LIN {X 0,Y 418.019,Z 608.172,A -85,B 0,C 180,E1 -10181.64,E2 -10181.64} C_VEL
LIN {X 0,Y 418.454,Z 601.286,A -85,B 0,C 180,E1 -10183.199,E2 -10183.199} C_VEL
LIN {X 0,Y 419.357,Z 591.379,A -85,B 0,C 180,E1 -10185.056,E2 -10185.056} C_VEL
LIN {X 0,Y 420.272,Z 581.997,A -85,B 0,C 180,E1 -10186.516,E2 -10186.516} C_VEL
LIN {X 0,Y 421.372,Z 571.359,A -85,B 0,C 180,E1 -10187.916,E2 -10187.916} C_VEL
LIN {X 0,Y 422.401,Z 559.979,A -85,B 0,C 180,E1 -10189.184,E2 -10189.184} C_VEL
LIN {X 0,Y 423.71,Z 546.942,A -85,B 0,C 180,E1 -10190.385,E2 -10190.385} C_VEL
LIN {X 0,Y 424.81,Z 534.302,A -85,B 0,C 180,E1 -10191.344,E2 -10191.344} C_VEL
LIN {X 0,Y 425.878,Z 520.707,A -85,B 0,C 180,E1 -10192.178,E2 -10192.178} C_VEL
LIN {X 0,Y 426.789,Z 506.169,A -85,B 0,C 180,E1 -10192.872,E2 -10192.872} C_VEL
LIN {X 0,Y 427.616,Z 490.972,A -85,B 0,C 180,E1 -10193.392,E2 -10193.392} C_VEL
LIN {X 0,Y 428.088,Z 474.732,A -85,B 0,C 180,E1 -10193.749,E2 -10193.749} C_VEL
LIN {X 0,Y 430.248,Z 350.197,A -85,B 0,C 180,E1 -10195.915,E2 -10195.915} C_VEL
LIN {X 0,Y 424.062,Z 318.078,A -85,B 0,C 180,E1 -10196.936,E2 -10196.936} C_VEL
LIN {X 0,Y 424.465,Z 312.588,A -85,B 0,C 180,E1 -10197.843,E2 -10197.843} C_VEL
LIN {X 0,Y 422.332,Z 302.144,A -85,B 0,C 180,E1 -10199.785,E2 -10199.785} C_VEL
LIN {X 0,Y 418.237,Z 286.016,A -85,B 0,C 180,E1 -10202.984,E2 -10202.984} C_VEL
LIN {X 0,Y 418.242,Z 286.015,A -85,B 0,C 180,E1 -10206.236,E2 -10206.236} C_VEL
LIN {X 0,Y 418.199,Z 286.022,A -85,B 0,C 180,E1 -10209.687,E2 -10209.687} C_VEL
LIN {X 0,Y 418.208,Z 286.015,A -85,B 0,C 180,E1 -10212.317,E2 -10212.317} C_VEL
LIN {X 0,Y 418.235,Z 286.012,A -85,B 0,C 180,E1 -10215.107,E2 -10215.107} C_VEL
LIN {X 0,Y 418.22,Z 286.015,A -85,B 0,C 180,E1 -10217.763,E2 -10217.763} C_VEL
LIN {X 0,Y 418.233,Z 286.01,A -85,B 0,C 180,E1 -10221.555,E2 -10221.555} C_VEL
LIN {X 0,Y 418.248,Z 286.005,A -85,B 0,C 180,E1 -10225.157,E2 -10225.157} C_VEL
LIN {X 0,Y 418.242,Z 286.009,A -85,B 0,C 180,E1 -10227.47,E2 -10227.47} C_VEL
LIN {X 0,Y 418.26,Z 286.007,A -85,B 0,C 180,E1 -10230.896,E2 -10230.896} C_VEL
LIN {X 0,Y 418.215,Z 286.019,A -85,B 0,C 180,E1 -10234.091,E2 -10234.091} C_VEL
LIN {X 0,Y 418.225,Z 286.012,A -85,B 0,C 180,E1 -10237.262,E2 -10237.262} C_VEL
LIN {X 0,Y 418.28,Z 286.004,A -85,B 0,C 180,E1 -10240.363,E2 -10240.363} C_VEL
LIN {X 0,Y 418.312,Z 286.006,A -85,B 0,C 180,E1 -10243.403,E2 -10243.403} C_VEL
LIN {X 0,Y 418.342,Z 285.979,A -85,B 0,C 180,E1 -10246.999,E2 -10246.999} C_VEL
LIN {X 0,Y 418.313,Z 285.998,A -85,B 0,C 180,E1 -10250.327,E2 -10250.327} C_VEL
LIN {X 0,Y 418.435,Z 285.988,A -85,B 0,C 180,E1 -10253.247,E2 -10253.247} C_VEL
LIN {X 0,Y 418.302,Z 285.996,A -85,B 0,C 180,E1 -10255.18,E2 -10255.18} C_VEL
LIN {X 0,Y 418.521,Z 285.966,A -85,B 0,C 180,E1 -10258.074,E2 -10258.074} C_VEL
LIN {X 0,Y 418.397,Z 285.989,A -85,B 0,C 180,E1 -10260.961,E2 -10260.961} C_VEL
LIN {X 0,Y 418.469,Z 285.98,A -85,B 0,C 180,E1 -10262.886,E2 -10262.886} C_VEL
LIN {X 0,Y 418.403,Z 285.965,A -85,B 0,C 180,E1 -10266.751,E2 -10266.751} C_VEL
LIN {X 0,Y 418.315,Z 286.001,A -85,B 0,C 180,E1 -10269.67,E2 -10269.67} C_VEL
LIN {X 0,Y 418.337,Z 285.999,A -85,B 0,C 180,E1 -10272.998,E2 -10272.998} C_VEL
LIN {X 0,Y 418.295,Z 285.982,A -85,B 0,C 180,E1 -10276.73,E2 -10276.73} C_VEL
LIN {X 0,Y 418.259,Z 286.005,A -85,B 0,C 180,E1 -10279.788,E2 -10279.788} C_VEL
LIN {X 0,Y 418.216,Z 286.013,A -85,B 0,C 180,E1 -10282.735,E2 -10282.735} C_VEL
LIN {X 0,Y 418.205,Z 285.997,A -85,B 0,C 180,E1 -10285.906,E2 -10285.906} C_VEL
LIN {X 0,Y 418.244,Z 286,A -85,B 0,C 180,E1 -10289.161,E2 -10289.161} C_VEL
LIN {X 0,Y 418.229,Z 286.011,A -85,B 0,C 180,E1 -10292.527,E2 -10292.527} C_VEL
LIN {X 0,Y 418.236,Z 286.006,A -85,B 0,C 180,E1 -10294.84,E2 -10294.84} C_VEL
LIN {X 0,Y 418.223,Z 286.002,A -85,B 0,C 180,E1 -10298.442,E2 -10298.442} C_VEL
LIN {X 0,Y 418.208,Z 286.013,A -85,B 0,C 180,E1 -10302.234,E2 -10302.234} C_VEL
LIN {X 0,Y 418.219,Z 286.001,A -85,B 0,C 180,E1 -10305.107,E2 -10305.107} C_VEL
LIN {X 0,Y 418.218,Z 286.012,A -85,B 0,C 180,E1 -10307.765,E2 -10307.765} C_VEL
LIN {X 0,Y 418.229,Z 286.015,A -85,B 0,C 180,E1 -10310.62,E2 -10310.62} C_VEL
LIN {X 0,Y 418.226,Z 286.004,A -85,B 0,C 180,E1 -10313.975,E2 -10313.975} C_VEL
LIN {X 0,Y 418.24,Z 286.012,A -85,B 0,C 180,E1 -10317.155,E2 -10317.155} C_VEL
LIN {X 0,Y 418.251,Z 286.006,A -85,B 0,C 180,E1 -10320.895,E2 -10320.895} C_VEL
LIN {X 0,Y 418.25,Z 286.006,A -85,B 0,C 180,E1 -10324.095,E2 -10324.095} C_VEL
LIN {X 0,Y 418.214,Z 286.016,A -85,B 0,C 180,E1 -10327.263,E2 -10327.263} C_VEL
LIN {X 0,Y 418.265,Z 286.004,A -85,B 0,C 180,E1 -10330.363,E2 -10330.363} C_VEL
LIN {X 0,Y 418.299,Z 285.999,A -85,B 0,C 180,E1 -10333.404,E2 -10333.404} C_VEL
LIN {X 0,Y 418.338,Z 285.999,A -85,B 0,C 180,E1 -10336.993,E2 -10336.993} C_VEL
LIN {X 0,Y 418.342,Z 285.997,A -85,B 0,C 180,E1 -10340.328,E2 -10340.328} C_VEL
LIN {X 0,Y 418.471,Z 285.983,A -85,B 0,C 180,E1 -10343.248,E2 -10343.248} C_VEL
LIN {X 0,Y 418.319,Z 286.004,A -85,B 0,C 180,E1 -10345.181,E2 -10345.181} C_VEL
LIN {X 0,Y 418.524,Z 285.974,A -85,B 0,C 180,E1 -10348.075,E2 -10348.075} C_VEL
LIN {X 0,Y 418.534,Z 285.982,A -85,B 0,C 180,E1 -10350.601,E2 -10350.601} C_VEL
LIN {X 0,Y 420.885,Z 296.753,A -85,B 0,C 180,E1 -10352.944,E2 -10352.944} C_VEL
LIN {X 0,Y 428.881,Z 316.026,A -85,B 0,C 180,E1 -10353.834,E2 -10353.834} C_VEL
LIN {X 0,Y 430.579,Z 324.35,A -85,B 0,C 180,E1 -10354.097,E2 -10354.097} C_VEL
LIN {X 0,Y 430.008,Z 354.65,A -85,B 0,C 180,E1 -10354.626,E2 -10354.626} C_VEL
LIN {X 0,Y 429.344,Z 360.497,A -85,B 0,C 180,E1 -10354.695,E2 -10354.695} C_VEL
LIN {X 0,Y 423.7,Z 379.54,A -85,B 0,C 180,E1 -10354.705,E2 -10354.705} C_VEL
LIN {X 0,Y 422.973,Z 385.393,A -85,B 0,C 180,E1 -10354.77,E2 -10354.77} C_VEL
LIN {X 0,Y 421.513,Z 462.7,A -85,B 0,C 180,E1 -10356.161,E2 -10356.161} C_VEL
LIN {X 0,Y 420.889,Z 477.855,A -85,B 0,C 180,E1 -10356.622,E2 -10356.622} C_VEL
LIN {X 0,Y 420.031,Z 492.733,A -85,B 0,C 180,E1 -10357.269,E2 -10357.269} C_VEL
LIN {X 0,Y 419.023,Z 507.308,A -85,B 0,C 180,E1 -10358.113,E2 -10358.113} C_VEL
LIN {X 0,Y 417.877,Z 520.501,A -85,B 0,C 180,E1 -10359.071,E2 -10359.071} C_VEL
LIN {X 0,Y 416.658,Z 533.182,A -85,B 0,C 180,E1 -10360.201,E2 -10360.201} C_VEL
LIN {X 0,Y 415.406,Z 545.864,A -85,B 0,C 180,E1 -10361.573,E2 -10361.573} C_VEL
LIN {X 0,Y 414.269,Z 556.742,A -85,B 0,C 180,E1 -10362.989,E2 -10362.989} C_VEL
LIN {X 0,Y 413.218,Z 566.322,A -85,B 0,C 180,E1 -10364.468,E2 -10364.468} C_VEL
LIN {X 0,Y 412.281,Z 575.139,A -85,B 0,C 180,E1 -10366.081,E2 -10366.081} C_VEL
LIN {X 0,Y 411.458,Z 583.427,A -85,B 0,C 180,E1 -10367.905,E2 -10367.905} C_VEL
LIN {X 0,Y 410.868,Z 590.526,A -85,B 0,C 180,E1 -10369.823,E2 -10369.823} C_VEL
LIN {X 0,Y 410.453,Z 595.842,A -85,B 0,C 180,E1 -10371.6,E2 -10371.6} C_VEL
LIN {X 0,Y 410.153,Z 600.738,A -85,B 0,C 180,E1 -10373.744,E2 -10373.744} C_VEL
LIN {X 0,Y 409.89,Z 603.462,A -85,B 0,C 180,E1 -10375.381,E2 -10375.381} C_VEL
LIN {X 0,Y 409.738,Z 605.849,A -85,B 0,C 180,E1 -10377.587,E2 -10377.587} C_VEL
LIN {X 0,Y 409.691,Z 606.635,A -85,B 0,C 180,E1 -10378.975,E2 -10378.975} C_VEL
LIN {X 0,Y 409.739,Z 606.704,A -85,B 0,C 180,E1 -10380.968,E2 -10380.968} C_VEL
LIN {X 0,Y 409.784,Z 605.724,A -85,B 0,C 180,E1 -10382.825,E2 -10382.825} C_VEL
LIN {X 0,Y 409.892,Z 603.843,A -85,B 0,C 180,E1 -10384.617,E2 -10384.617} C_VEL
LIN {X 0,Y 410.153,Z 601.026,A -85,B 0,C 180,E1 -10386.36,E2 -10386.36} C_VEL
LIN {X 0,Y 410.415,Z 597.353,A -85,B 0,C 180,E1 -10388.057,E2 -10388.057} C_VEL
LIN {X 0,Y 410.855,Z 591.79,A -85,B 0,C 180,E1 -10390.053,E2 -10390.053} C_VEL
LIN {X 0,Y 411.509,Z 584.791,A -85,B 0,C 180,E1 -10392.028,E2 -10392.028} C_VEL
LIN {X 0,Y 412.221,Z 577.732,A -85,B 0,C 180,E1 -10393.667,E2 -10393.667} C_VEL
LIN {X 0,Y 413.095,Z 569.526,A -85,B 0,C 180,E1 -10395.257,E2 -10395.257} C_VEL
LIN {X 0,Y 414.171,Z 559.721,A -85,B 0,C 180,E1 -10396.856,E2 -10396.856} C_VEL
LIN {X 0,Y 415.357,Z 549.189,A -85,B 0,C 180,E1 -10398.296,E2 -10398.296} C_VEL
LIN {X 0,Y 416.685,Z 536.811,A -85,B 0,C 180,E1 -10399.709,E2 -10399.709} C_VEL
LIN {X 0,Y 417.964,Z 524.647,A -85,B 0,C 180,E1 -10400.856,E2 -10400.856} C_VEL
LIN {X 0,Y 419.116,Z 511.674,A -85,B 0,C 180,E1 -10401.868,E2 -10401.868} C_VEL
LIN {X 0,Y 420.267,Z 497.228,A -85,B 0,C 180,E1 -10402.766,E2 -10402.766} C_VEL
LIN {X 0,Y 421.236,Z 482.096,A -85,B 0,C 180,E1 -10403.483,E2 -10403.483} C_VEL
LIN {X 0,Y 421.955,Z 466.599,A -85,B 0,C 180,E1 -10404.006,E2 -10404.006} C_VEL
LIN {X 0,Y 422.457,Z 446.837,A -85,B 0,C 180,E1 -10404.418,E2 -10404.418} C_VEL
LIN {X 0,Y 424.854,Z 325.118,A -85,B 0,C 180,E1 -10406.598,E2 -10406.598} C_VEL
LIN {X 0,Y 423.221,Z 318.56,A -85,B 0,C 180,E1 -10406.844,E2 -10406.844} C_VEL
LIN {X 0,Y 415.127,Z 300.427,A -85,B 0,C 180,E1 -10407.818,E2 -10407.818} C_VEL
LIN {X 0,Y 413.924,Z 297.657,A -85,B 0,C 180,E1 -10408.001,E2 -10408.001} C_VEL
LIN {X 0,Y 411.237,Z 286.889,A -85,B 0,C 180,E1 -10410.516,E2 -10410.516} C_VEL
LIN {X 0,Y 411.222,Z 286.886,A -85,B 0,C 180,E1 -10413.62,E2 -10413.62} C_VEL
LIN {X 0,Y 411.188,Z 286.896,A -85,B 0,C 180,E1 -10416.854,E2 -10416.854} C_VEL
LIN {X 0,Y 411.2,Z 286.89,A -85,B 0,C 180,E1 -10420.052,E2 -10420.052} C_VEL
LIN {X 0,Y 411.249,Z 286.886,A -85,B 0,C 180,E1 -10423.133,E2 -10423.133} C_VEL
LIN {X 0,Y 411.291,Z 286.879,A -85,B 0,C 180,E1 -10426.898,E2 -10426.898} C_VEL
LIN {X 0,Y 411.279,Z 286.878,A -85,B 0,C 180,E1 -10430.163,E2 -10430.163} C_VEL
LIN {X 0,Y 411.445,Z 286.859,A -85,B 0,C 180,E1 -10433.135,E2 -10433.135} C_VEL
LIN {X 0,Y 411.295,Z 286.88,A -85,B 0,C 180,E1 -10435.101,E2 -10435.101} C_VEL
LIN {X 0,Y 411.5,Z 286.85,A -85,B 0,C 180,E1 -10438.044,E2 -10438.044} C_VEL
LIN {X 0,Y 411.629,Z 286.833,A -85,B 0,C 180,E1 -10440.002,E2 -10440.002} C_VEL
LIN {X 0,Y 411.442,Z 286.86,A -85,B 0,C 180,E1 -10442.939,E2 -10442.939} C_VEL
LIN {X 0,Y 411.423,Z 286.862,A -85,B 0,C 180,E1 -10446.869,E2 -10446.869} C_VEL
LIN {X 0,Y 411.28,Z 286.877,A -85,B 0,C 180,E1 -10449.84,E2 -10449.84} C_VEL
LIN {X 0,Y 411.297,Z 286.875,A -85,B 0,C 180,E1 -10453.105,E2 -10453.105} C_VEL
LIN {X 0,Y 411.249,Z 286.88,A -85,B 0,C 180,E1 -10456.89,E2 -10456.89} C_VEL
LIN {X 0,Y 411.223,Z 286.884,A -85,B 0,C 180,E1 -10459.988,E2 -10459.988} C_VEL
LIN {X 0,Y 411.179,Z 286.888,A -85,B 0,C 180,E1 -10463.15,E2 -10463.15} C_VEL
LIN {X 0,Y 411.167,Z 286.891,A -85,B 0,C 180,E1 -10466.387,E2 -10466.387} C_VEL
LIN {X 0,Y 411.19,Z 286.886,A -85,B 0,C 180,E1 -10469.715,E2 -10469.715} C_VEL
LIN {X 0,Y 411.199,Z 286.886,A -85,B 0,C 180,E1 -10473.158,E2 -10473.158} C_VEL
LIN {X 0,Y 411.183,Z 286.888,A -85,B 0,C 180,E1 -10476.553,E2 -10476.553} C_VEL
LIN {X 0,Y 411.163,Z 286.89,A -85,B 0,C 180,E1 -10479.721,E2 -10479.721} C_VEL
LIN {X 0,Y 411.158,Z 286.892,A -85,B 0,C 180,E1 -10483.137,E2 -10483.137} C_VEL
LIN {X 0,Y 411.16,Z 286.894,A -85,B 0,C 180,E1 -10485.883,E2 -10485.883} C_VEL
LIN {X 0,Y 411.155,Z 286.894,A -85,B 0,C 180,E1 -10489.494,E2 -10489.494} C_VEL
LIN {X 0,Y 411.179,Z 286.892,A -85,B 0,C 180,E1 -10492.026,E2 -10492.026} C_VEL
LIN {X 0,Y 411.202,Z 286.885,A -85,B 0,C 180,E1 -10495.667,E2 -10495.667} C_VEL
LIN {X 0,Y 411.239,Z 286.989,A -85,B 0,C 180,E1 -10496.262,E2 -10496.262} C_VEL
LIN {X 0,Y 415.258,Z 302.312,A -85,B 0,C 180,E1 -10499.488,E2 -10499.488} C_VEL
LIN {X 0,Y 417.681,Z 313.276,A -85,B 0,C 180,E1 -10501.653,E2 -10501.653} C_VEL
LIN {X 0,Y 417.681,Z 317.189,A -85,B 0,C 180,E1 -10502.344,E2 -10502.344} C_VEL
LIN {X 0,Y 422.839,Z 342.545,A -85,B 0,C 180,E1 -10503.237,E2 -10503.237} C_VEL
LIN {X 0,Y 424.557,Z 352.473,A -85,B 0,C 180,E1 -10503.551,E2 -10503.551} C_VEL
LIN {X 0,Y 421.834,Z 483.858,A -85,B 0,C 180,E1 -10505.91,E2 -10505.91} C_VEL
LIN {X 0,Y 421.04,Z 499.798,A -85,B 0,C 180,E1 -10506.385,E2 -10506.385} C_VEL
LIN {X 0,Y 420.117,Z 514.266,A -85,B 0,C 180,E1 -10507.007,E2 -10507.007} C_VEL
LIN {X 0,Y 418.915,Z 528.72,A -85,B 0,C 180,E1 -10507.824,E2 -10507.824} C_VEL
LIN {X 0,Y 417.691,Z 542.21,A -85,B 0,C 180,E1 -10508.793,E2 -10508.793} C_VEL
LIN {X 0,Y 416.259,Z 555.968,A -85,B 0,C 180,E1 -10510.008,E2 -10510.008} C_VEL
LIN {X 0,Y 415.097,Z 567.363,A -85,B 0,C 180,E1 -10511.236,E2 -10511.236} C_VEL
LIN {X 0,Y 413.886,Z 578.907,A -85,B 0,C 180,E1 -10512.714,E2 -10512.714} C_VEL
LIN {X 0,Y 412.782,Z 588.63,A -85,B 0,C 180,E1 -10514.193,E2 -10514.193} C_VEL
LIN {X 0,Y 411.805,Z 598.188,A -85,B 0,C 180,E1 -10515.926,E2 -10515.926} C_VEL
LIN {X 0,Y 411.112,Z 606.159,A -85,B 0,C 180,E1 -10517.662,E2 -10517.662} C_VEL
LIN {X 0,Y 410.504,Z 613.606,A -85,B 0,C 180,E1 -10519.645,E2 -10519.645} C_VEL
LIN {X 0,Y 410.2,Z 619.523,A -85,B 0,C 180,E1 -10521.627,E2 -10521.627} C_VEL
LIN {X 0,Y 410.012,Z 623.044,A -85,B 0,C 180,E1 -10523.109,E2 -10523.109} C_VEL
LIN {X 0,Y 409.927,Z 626.598,A -85,B 0,C 180,E1 -10525.083,E2 -10525.083} C_VEL
LIN {X 0,Y 409.906,Z 628.934,A -85,B 0,C 180,E1 -10527.052,E2 -10527.052} C_VEL
LIN {X 0,Y 409.935,Z 630.103,A -85,B 0,C 180,E1 -10529.018,E2 -10529.018} C_VEL
LIN {X 0,Y 409.935,Z 630.105,A -85,B 0,C 180,E1 -10530.983,E2 -10530.983} C_VEL
LIN {X 0,Y 409.907,Z 628.9,A -85,B 0,C 180,E1 -10532.949,E2 -10532.949} C_VEL
LIN {X 0,Y 409.935,Z 626.527,A -85,B 0,C 180,E1 -10534.918,E2 -10534.918} C_VEL
LIN {X 0,Y 410.051,Z 622.935,A -85,B 0,C 180,E1 -10536.891,E2 -10536.891} C_VEL
LIN {X 0,Y 410.241,Z 618.028,A -85,B 0,C 180,E1 -10538.87,E2 -10538.87} C_VEL
LIN {X 0,Y 410.674,Z 611.68,A -85,B 0,C 180,E1 -10540.851,E2 -10540.851} C_VEL
LIN {X 0,Y 411.254,Z 603.708,A -85,B 0,C 180,E1 -10542.836,E2 -10542.836} C_VEL
LIN {X 0,Y 412.049,Z 595.217,A -85,B 0,C 180,E1 -10544.571,E2 -10544.571} C_VEL
LIN {X 0,Y 412.824,Z 586.588,A -85,B 0,C 180,E1 -10546.06,E2 -10546.06} C_VEL
LIN {X 0,Y 414.02,Z 576.388,A -85,B 0,C 180,E1 -10547.536,E2 -10547.536} C_VEL
LIN {X 0,Y 415.067,Z 565.321,A -85,B 0,C 180,E1 -10548.895,E2 -10548.895} C_VEL
LIN {X 0,Y 416.3,Z 553.387,A -85,B 0,C 180,E1 -10550.119,E2 -10550.119} C_VEL
LIN {X 0,Y 417.551,Z 540.482,A -85,B 0,C 180,E1 -10551.215,E2 -10551.215} C_VEL
LIN {X 0,Y 418.753,Z 526.377,A -85,B 0,C 180,E1 -10552.186,E2 -10552.186} C_VEL
LIN {X 0,Y 419.881,Z 511.447,A -85,B 0,C 180,E1 -10552.986,E2 -10552.986} C_VEL
LIN {X 0,Y 420.719,Z 496.663,A -85,B 0,C 180,E1 -10553.575,E2 -10553.575} C_VEL
LIN {X 0,Y 421.368,Z 481.331,A -85,B 0,C 180,E1 -10553.988,E2 -10553.988} C_VEL
LIN {X 0,Y 423.834,Z 353.002,A -85,B 0,C 180,E1 -10556.261,E2 -10556.261} C_VEL
LIN {X 0,Y 423.233,Z 348.315,A -85,B 0,C 180,E1 -10556.388,E2 -10556.388} C_VEL
LIN {X 0,Y 417.369,Z 317.942,A -85,B 0,C 180,E1 -10557.375,E2 -10557.375} C_VEL
LIN {X 0,Y 417.596,Z 313.587,A -85,B 0,C 180,E1 -10558.114,E2 -10558.114} C_VEL
LIN {X 0,Y 414.758,Z 300.84,A -85,B 0,C 180,E1 -10560.553,E2 -10560.553} C_VEL
LIN {X 0,Y 411.192,Z 286.894,A -85,B 0,C 180,E1 -10563.369,E2 -10563.369} C_VEL
LIN {X 0,Y 411.188,Z 286.896,A -85,B 0,C 180,E1 -10566.742,E2 -10566.742} C_VEL
LIN {X 0,Y 411.169,Z 286.897,A -85,B 0,C 180,E1 -10569.719,E2 -10569.719} C_VEL
LIN {X 0,Y 411.162,Z 286.889,A -85,B 0,C 180,E1 -10573.134,E2 -10573.134} C_VEL
LIN {X 0,Y 411.164,Z 286.893,A -85,B 0,C 180,E1 -10575.881,E2 -10575.881} C_VEL
LIN {X 0,Y 411.148,Z 286.898,A -85,B 0,C 180,E1 -10578.773,E2 -10578.773} C_VEL
LIN {X 0,Y 411.18,Z 286.894,A -85,B 0,C 180,E1 -10582.024,E2 -10582.024} C_VEL
LIN {X 0,Y 411.2,Z 286.883,A -85,B 0,C 180,E1 -10585.123,E2 -10585.123} C_VEL
LIN {X 0,Y 411.163,Z 286.897,A -85,B 0,C 180,E1 -10588.001,E2 -10588.001} C_VEL
LIN {X 0,Y 411.174,Z 286.892,A -85,B 0,C 180,E1 -10591.405,E2 -10591.405} C_VEL
LIN {X 0,Y 411.186,Z 286.891,A -85,B 0,C 180,E1 -10594.94,E2 -10594.94} C_VEL
LIN {X 0,Y 411.2,Z 286.895,A -85,B 0,C 180,E1 -10597.912,E2 -10597.912} C_VEL
LIN {X 0,Y 411.214,Z 286.884,A -85,B 0,C 180,E1 -10601.05,E2 -10601.05} C_VEL
LIN {X 0,Y 411.247,Z 286.88,A -85,B 0,C 180,E1 -10604.13,E2 -10604.13} C_VEL
LIN {X 0,Y 411.297,Z 286.855,A -85,B 0,C 180,E1 -10607.164,E2 -10607.164} C_VEL
LIN {X 0,Y 411.268,Z 286.877,A -85,B 0,C 180,E1 -10610.159,E2 -10610.159} C_VEL
LIN {X 0,Y 411.384,Z 286.865,A -85,B 0,C 180,E1 -10613.13,E2 -10613.13} C_VEL
LIN {X 0,Y 411.274,Z 286.872,A -85,B 0,C 180,E1 -10615.097,E2 -10615.097} C_VEL
LIN {X 0,Y 411.49,Z 286.84,A -85,B 0,C 180,E1 -10618.041,E2 -10618.041} C_VEL
LIN {X 0,Y 411.497,Z 286.85,A -85,B 0,C 180,E1 -10621.956,E2 -10621.956} C_VEL
LIN {X 0,Y 411.348,Z 286.843,A -85,B 0,C 180,E1 -10626.445,E2 -10626.445} C_VEL
LIN {X 0,Y 411.276,Z 286.867,A -85,B 0,C 180,E1 -10628.845,E2 -10628.845} C_VEL
LIN {X 0,Y 411.271,Z 286.879,A -85,B 0,C 180,E1 -10631.831,E2 -10631.831} C_VEL
LIN {X 0,Y 411.237,Z 286.876,A -85,B 0,C 180,E1 -10634.852,E2 -10634.852} C_VEL
LIN {X 0,Y 411.23,Z 286.868,A -85,B 0,C 180,E1 -10637.914,E2 -10637.914} C_VEL
LIN {X 0,Y 411.185,Z 286.888,A -85,B 0,C 180,E1 -10641.033,E2 -10641.033} C_VEL
LIN {X 0,Y 411.178,Z 286.884,A -85,B 0,C 180,E1 -10644.216,E2 -10644.216} C_VEL
LIN {X 0,Y 411.133,Z 286.876,A -85,B 0,C 180,E1 -10647.484,E2 -10647.484} C_VEL
LIN {X 0,Y 411.183,Z 286.886,A -85,B 0,C 180,E1 -10649.712,E2 -10649.712} C_VEL
LIN {X 0,Y 411.191,Z 286.89,A -85,B 0,C 180,E1 -10653.155,E2 -10653.155} C_VEL
LIN {X 0,Y 411.177,Z 286.872,A -85,B 0,C 180,E1 -10656.551,E2 -10656.551} C_VEL
LIN {X 0,Y 411.155,Z 286.892,A -85,B 0,C 180,E1 -10659.719,E2 -10659.719} C_VEL
LIN {X 0,Y 411.149,Z 286.891,A -85,B 0,C 180,E1 -10663.134,E2 -10663.134} C_VEL
LIN {X 0,Y 411.15,Z 286.881,A -85,B 0,C 180,E1 -10665.88,E2 -10665.88} C_VEL
LIN {X 0,Y 411.144,Z 286.897,A -85,B 0,C 180,E1 -10668.771,E2 -10668.771} C_VEL
LIN {X 0,Y 411.175,Z 286.883,A -85,B 0,C 180,E1 -10672.025,E2 -10672.025} C_VEL
LIN {X 0,Y 411.188,Z 286.889,A -85,B 0,C 180,E1 -10675.665,E2 -10675.665} C_VEL
LIN {X 0,Y 411.172,Z 286.882,A -85,B 0,C 180,E1 -10679.151,E2 -10679.151} C_VEL
LIN {X 0,Y 411.249,Z 286.885,A -85,B 0,C 180,E1 -10682.698,E2 -10682.698} C_VEL
LIN {X 0,Y 411.194,Z 286.884,A -85,B 0,C 180,E1 -10685.783,E2 -10685.783} C_VEL
LIN {X 0,Y 411.179,Z 286.887,A -85,B 0,C 180,E1 -10688.965,E2 -10688.965} C_VEL
LIN {X 0,Y 411.234,Z 286.885,A -85,B 0,C 180,E1 -10692.084,E2 -10692.084} C_VEL
LIN {X 0,Y 411.244,Z 286.884,A -85,B 0,C 180,E1 -10695.147,E2 -10695.147} C_VEL
LIN {X 0,Y 411.283,Z 286.879,A -85,B 0,C 180,E1 -10698.167,E2 -10698.167} C_VEL
LIN {X 0,Y 411.422,Z 286.859,A -85,B 0,C 180,E1 -10702.188,E2 -10702.188} C_VEL
LIN {X 0,Y 411.452,Z 286.857,A -85,B 0,C 180,E1 -10704.117,E2 -10704.117} C_VEL
LIN {X 0,Y 411.493,Z 286.85,A -85,B 0,C 180,E1 -10708.042,E2 -10708.042} C_VEL
LIN {X 0,Y 411.583,Z 286.917,A -85,B 0,C 180,E1 -10710.275,E2 -10710.275} C_VEL
LIN {X 0,Y 413.798,Z 296.991,A -85,B 0,C 180,E1 -10712.464,E2 -10712.464} C_VEL
LIN {X 0,Y 422.753,Z 318.435,A -85,B 0,C 180,E1 -10713.484,E2 -10713.484} C_VEL
LIN {X 0,Y 424.172,Z 324.99,A -85,B 0,C 180,E1 -10713.701,E2 -10713.701} C_VEL
LIN {X 0,Y 422.973,Z 385.393,A -85,B 0,C 180,E1 -10714.77,E2 -10714.77} C_VEL
LIN {X 0,Y 422.255,Z 391.242,A -85,B 0,C 180,E1 -10714.835,E2 -10714.835} C_VEL
LIN {X 0,Y 416.637,Z 410.284,A -85,B 0,C 180,E1 -10714.849,E2 -10714.849} C_VEL
LIN {X 0,Y 415.934,Z 416.132,A -85,B 0,C 180,E1 -10714.917,E2 -10714.917} C_VEL
LIN {X 0,Y 415.006,Z 462.388,A -85,B 0,C 180,E1 -10715.77,E2 -10715.77} C_VEL
LIN {X 0,Y 414.361,Z 477.695,A -85,B 0,C 180,E1 -10716.237,E2 -10716.237} C_VEL
LIN {X 0,Y 413.461,Z 492.672,A -85,B 0,C 180,E1 -10716.894,E2 -10716.894} C_VEL
LIN {X 0,Y 412.448,Z 506.704,A -85,B 0,C 180,E1 -10717.711,E2 -10717.711} C_VEL
LIN {X 0,Y 411.177,Z 520.857,A -85,B 0,C 180,E1 -10718.749,E2 -10718.749} C_VEL
LIN {X 0,Y 409.817,Z 534.542,A -85,B 0,C 180,E1 -10719.999,E2 -10719.999} C_VEL
LIN {X 0,Y 408.552,Z 546.595,A -85,B 0,C 180,E1 -10721.34,E2 -10721.34} C_VEL
LIN {X 0,Y 407.239,Z 558.65,A -85,B 0,C 180,E1 -10722.964,E2 -10722.964} C_VEL
LIN {X 0,Y 406.076,Z 568.746,A -85,B 0,C 180,E1 -10724.598,E2 -10724.598} C_VEL
LIN {X 0,Y 405.06,Z 577.869,A -85,B 0,C 180,E1 -10726.376,E2 -10726.376} C_VEL
LIN {X 0,Y 404.281,Z 585.722,A -85,B 0,C 180,E1 -10728.234,E2 -10728.234} C_VEL
LIN {X 0,Y 403.752,Z 591.697,A -85,B 0,C 180,E1 -10729.963,E2 -10729.963} C_VEL
LIN {X 0,Y 403.315,Z 597.333,A -85,B 0,C 180,E1 -10731.988,E2 -10731.988} C_VEL
LIN {X 0,Y 403.095,Z 600.926,A -85,B 0,C 180,E1 -10733.64,E2 -10733.64} C_VEL
LIN {X 0,Y 402.742,Z 604.399,A -85,B 0,C 180,E1 -10735.864,E2 -10735.864} C_VEL
LIN {X 0,Y 402.697,Z 605.701,A -85,B 0,C 180,E1 -10737.124,E2 -10737.124} C_VEL
LIN {X 0,Y 402.584,Z 606.898,A -85,B 0,C 180,E1 -10739.261,E2 -10739.261} C_VEL
LIN {X 0,Y 402.632,Z 606.873,A -85,B 0,C 180,E1 -10741.212,E2 -10741.212} C_VEL
LIN {X 0,Y 402.7,Z 605.756,A -85,B 0,C 180,E1 -10743.106,E2 -10743.106} C_VEL
LIN {X 0,Y 402.867,Z 603.424,A -85,B 0,C 180,E1 -10745.146,E2 -10745.146} C_VEL
LIN {X 0,Y 403.136,Z 600.871,A -85,B 0,C 180,E1 -10746.689,E2 -10746.689} C_VEL
LIN {X 0,Y 403.505,Z 596.049,A -85,B 0,C 180,E1 -10748.829,E2 -10748.829} C_VEL
LIN {X 0,Y 403.968,Z 590.478,A -85,B 0,C 180,E1 -10750.721,E2 -10750.721} C_VEL
LIN {X 0,Y 404.711,Z 583.498,A -85,B 0,C 180,E1 -10752.628,E2 -10752.628} C_VEL
LIN {X 0,Y 405.604,Z 574.901,A -85,B 0,C 180,E1 -10754.544,E2 -10754.544} C_VEL
LIN {X 0,Y 406.742,Z 565.413,A -85,B 0,C 180,E1 -10756.282,E2 -10756.282} C_VEL
LIN {X 0,Y 407.897,Z 555.484,A -85,B 0,C 180,E1 -10757.805,E2 -10757.805} C_VEL
LIN {X 0,Y 409.259,Z 544.082,A -85,B 0,C 180,E1 -10759.269,E2 -10759.269} C_VEL
LIN {X 0,Y 410.653,Z 531.345,A -85,B 0,C 180,E1 -10760.627,E2 -10760.627} C_VEL
LIN {X 0,Y 412.046,Z 517.625,A -85,B 0,C 180,E1 -10761.82,E2 -10761.82} C_VEL
LIN {X 0,Y 413.242,Z 504.086,A -85,B 0,C 180,E1 -10762.768,E2 -10762.768} C_VEL
LIN {X 0,Y 414.345,Z 489.154,A -85,B 0,C 180,E1 -10763.586,E2 -10763.586} C_VEL
LIN {X 0,Y 415.232,Z 473.83,A -85,B 0,C 180,E1 -10764.203,E2 -10764.203} C_VEL
LIN {X 0,Y 415.815,Z 458.836,A -85,B 0,C 180,E1 -10764.61,E2 -10764.61} C_VEL
LIN {X 0,Y 418.589,Z 326.369,A -85,B 0,C 180,E1 -10767.031,E2 -10767.031} C_VEL
LIN {X 0,Y 417.293,Z 321.295,A -85,B 0,C 180,E1 -10767.23,E2 -10767.23} C_VEL
LIN {X 0,Y 409.485,Z 303.858,A -85,B 0,C 180,E1 -10768.195,E2 -10768.195} C_VEL
LIN {X 0,Y 406.781,Z 297.955,A -85,B 0,C 180,E1 -10768.566,E2 -10768.566} C_VEL
LIN {X 0,Y 404.175,Z 287.765,A -85,B 0,C 180,E1 -10771.009,E2 -10771.009} C_VEL
LIN {X 0,Y 404.168,Z 287.767,A -85,B 0,C 180,E1 -10774.235,E2 -10774.235} C_VEL
LIN {X 0,Y 404.155,Z 287.766,A -85,B 0,C 180,E1 -10777.51,E2 -10777.51} C_VEL
LIN {X 0,Y 404.151,Z 287.764,A -85,B 0,C 180,E1 -10780.709,E2 -10780.709} C_VEL
LIN {X 0,Y 404.207,Z 287.762,A -85,B 0,C 180,E1 -10783.85,E2 -10783.85} C_VEL
LIN {X 0,Y 404.269,Z 287.753,A -85,B 0,C 180,E1 -10786.94,E2 -10786.94} C_VEL
LIN {X 0,Y 404.244,Z 287.754,A -85,B 0,C 180,E1 -10789.99,E2 -10789.99} C_VEL
LIN {X 0,Y 404.392,Z 287.739,A -85,B 0,C 180,E1 -10793.014,E2 -10793.014} C_VEL
LIN {X 0,Y 404.268,Z 287.755,A -85,B 0,C 180,E1 -10795.015,E2 -10795.015} C_VEL
LIN {X 0,Y 404.468,Z 287.726,A -85,B 0,C 180,E1 -10798.01,E2 -10798.01} C_VEL
LIN {X 0,Y 404.599,Z 287.709,A -85,B 0,C 180,E1 -10800.002,E2 -10800.002} C_VEL
LIN {X 0,Y 404.4,Z 287.738,A -85,B 0,C 180,E1 -10802.99,E2 -10802.99} C_VEL
LIN {X 0,Y 404.373,Z 287.738,A -85,B 0,C 180,E1 -10806.989,E2 -10806.989} C_VEL
LIN {X 0,Y 404.241,Z 287.753,A -85,B 0,C 180,E1 -10811.027,E2 -10811.027} C_VEL
LIN {X 0,Y 404.201,Z 287.757,A -85,B 0,C 180,E1 -10814.09,E2 -10814.09} C_VEL
LIN {X 0,Y 404.195,Z 287.758,A -85,B 0,C 180,E1 -10817.194,E2 -10817.194} C_VEL
LIN {X 0,Y 404.156,Z 287.764,A -85,B 0,C 180,E1 -10820.353,E2 -10820.353} C_VEL
LIN {X 0,Y 404.141,Z 287.764,A -85,B 0,C 180,E1 -10823.578,E2 -10823.578} C_VEL
LIN {X 0,Y 404.113,Z 287.772,A -85,B 0,C 180,E1 -10826.884,E2 -10826.884} C_VEL
LIN {X 0,Y 404.137,Z 287.77,A -85,B 0,C 180,E1 -10830.287,E2 -10830.287} C_VEL
LIN {X 0,Y 404.132,Z 287.768,A -85,B 0,C 180,E1 -10833.815,E2 -10833.815} C_VEL
LIN {X 0,Y 404.125,Z 287.767,A -85,B 0,C 180,E1 -10836.875,E2 -10836.875} C_VEL
LIN {X 0,Y 404.113,Z 287.772,A -85,B 0,C 180,E1 -10840.076,E2 -10840.076} C_VEL
LIN {X 0,Y 404.137,Z 287.767,A -85,B 0,C 180,E1 -10843.083,E2 -10843.083} C_VEL
LIN {X 0,Y 404.117,Z 287.771,A -85,B 0,C 180,E1 -10845.923,E2 -10845.923} C_VEL
LIN {X 0,Y 404.099,Z 287.774,A -85,B 0,C 180,E1 -10848.634,E2 -10848.634} C_VEL
LIN {X 0,Y 404.135,Z 287.772,A -85,B 0,C 180,E1 -10851.497,E2 -10851.497} C_VEL
LIN {X 0,Y 404.18,Z 287.761,A -85,B 0,C 180,E1 -10854.985,E2 -10854.985} C_VEL
LIN {X 0,Y 404.182,Z 287.789,A -85,B 0,C 180,E1 -10855.742,E2 -10855.742} C_VEL
LIN {X 0,Y 408.316,Z 303.343,A -85,B 0,C 180,E1 -10859.113,E2 -10859.113} C_VEL
LIN {X 0,Y 410.827,Z 314.595,A -85,B 0,C 180,E1 -10861.381,E2 -10861.381} C_VEL
LIN {X 0,Y 411.081,Z 317.033,A -85,B 0,C 180,E1 -10861.841,E2 -10861.841} C_VEL
LIN {X 0,Y 416.364,Z 342.596,A -85,B 0,C 180,E1 -10862.766,E2 -10862.766} C_VEL
LIN {X 0,Y 418.219,Z 354.039,A -85,B 0,C 180,E1 -10863.131,E2 -10863.131} C_VEL
LIN {X 0,Y 415.424,Z 482.982,A -85,B 0,C 180,E1 -10865.481,E2 -10865.481} C_VEL
LIN {X 0,Y 414.6,Z 499.2,A -85,B 0,C 180,E1 -10865.962,E2 -10865.962} C_VEL
LIN {X 0,Y 413.669,Z 512.956,A -85,B 0,C 180,E1 -10866.555,E2 -10866.555} C_VEL
LIN {X 0,Y 412.49,Z 526.752,A -85,B 0,C 180,E1 -10867.327,E2 -10867.327} C_VEL
LIN {X 0,Y 411.221,Z 540.575,A -85,B 0,C 180,E1 -10868.311,E2 -10868.311} C_VEL
LIN {X 0,Y 409.857,Z 553.279,A -85,B 0,C 180,E1 -10869.42,E2 -10869.42} C_VEL
LIN {X 0,Y 408.489,Z 565.084,A -85,B 0,C 180,E1 -10870.66,E2 -10870.66} C_VEL
LIN {X 0,Y 407.212,Z 576.972,A -85,B 0,C 180,E1 -10872.162,E2 -10872.162} C_VEL
LIN {X 0,Y 406.021,Z 586.982,A -85,B 0,C 180,E1 -10873.664,E2 -10873.664} C_VEL
LIN {X 0,Y 404.969,Z 596.786,A -85,B 0,C 180,E1 -10875.426,E2 -10875.426} C_VEL
LIN {X 0,Y 404.203,Z 604.974,A -85,B 0,C 180,E1 -10877.192,E2 -10877.192} C_VEL
LIN {X 0,Y 403.658,Z 611.756,A -85,B 0,C 180,E1 -10878.959,E2 -10878.959} C_VEL
LIN {X 0,Y 403.18,Z 618.015,A -85,B 0,C 180,E1 -10880.975,E2 -10880.975} C_VEL
LIN {X 0,Y 402.926,Z 622.858,A -85,B 0,C 180,E1 -10882.987,E2 -10882.987} C_VEL
LIN {X 0,Y 402.84,Z 626.406,A -85,B 0,C 180,E1 -10884.996,E2 -10884.996} C_VEL
LIN {X 0,Y 402.804,Z 628.737,A -85,B 0,C 180,E1 -10887,E2 -10887} C_VEL
LIN {X 0,Y 402.862,Z 629.902,A -85,B 0,C 180,E1 -10889.001,E2 -10889.001} C_VEL
LIN {X 0,Y 402.862,Z 629.9,A -85,B 0,C 180,E1 -10891,E2 -10891} C_VEL
LIN {X 0,Y 402.805,Z 628.688,A -85,B 0,C 180,E1 -10893.001,E2 -10893.001} C_VEL
LIN {X 0,Y 402.852,Z 626.308,A -85,B 0,C 180,E1 -10895.004,E2 -10895.004} C_VEL
LIN {X 0,Y 402.973,Z 622.705,A -85,B 0,C 180,E1 -10897.013,E2 -10897.013} C_VEL
LIN {X 0,Y 403.185,Z 617.788,A -85,B 0,C 180,E1 -10899.026,E2 -10899.026} C_VEL
LIN {X 0,Y 403.631,Z 611.426,A -85,B 0,C 180,E1 -10901.042,E2 -10901.042} C_VEL
LIN {X 0,Y 404.21,Z 603.431,A -85,B 0,C 180,E1 -10903.064,E2 -10903.064} C_VEL
LIN {X 0,Y 405.107,Z 594.918,A -85,B 0,C 180,E1 -10904.826,E2 -10904.826} C_VEL
LIN {X 0,Y 405.913,Z 586.269,A -85,B 0,C 180,E1 -10906.341,E2 -10906.341} C_VEL
LIN {X 0,Y 407.188,Z 576.038,A -85,B 0,C 180,E1 -10907.84,E2 -10907.84} C_VEL
LIN {X 0,Y 408.293,Z 564.94,A -85,B 0,C 180,E1 -10909.22,E2 -10909.22} C_VEL
LIN {X 0,Y 409.54,Z 552.964,A -85,B 0,C 180,E1 -10910.466,E2 -10910.466} C_VEL
LIN {X 0,Y 410.905,Z 540.012,A -85,B 0,C 180,E1 -10911.576,E2 -10911.576} C_VEL
LIN {X 0,Y 412.155,Z 525.838,A -85,B 0,C 180,E1 -10912.561,E2 -10912.561} C_VEL
LIN {X 0,Y 413.237,Z 512.176,A -85,B 0,C 180,E1 -10913.307,E2 -10913.307} C_VEL
LIN {X 0,Y 414.099,Z 497.808,A -85,B 0,C 180,E1 -10913.904,E2 -10913.904} C_VEL
LIN {X 0,Y 414.781,Z 483.107,A -85,B 0,C 180,E1 -10914.327,E2 -10914.327} C_VEL
LIN {X 0,Y 417.4,Z 354.08,A -85,B 0,C 180,E1 -10916.653,E2 -10916.653} C_VEL
LIN {X 0,Y 417.074,Z 350.968,A -85,B 0,C 180,E1 -10916.735,E2 -10916.735} C_VEL
LIN {X 0,Y 410.676,Z 317.785,A -85,B 0,C 180,E1 -10917.832,E2 -10917.832} C_VEL
LIN {X 0,Y 410.712,Z 314.837,A -85,B 0,C 180,E1 -10918.349,E2 -10918.349} C_VEL
LIN {X 0,Y 407.689,Z 301.514,A -85,B 0,C 180,E1 -10920.956,E2 -10920.956} C_VEL
LIN {X 0,Y 404.172,Z 287.765,A -85,B 0,C 180,E1 -10923.809,E2 -10923.809} C_VEL
LIN {X 0,Y 404.135,Z 287.773,A -85,B 0,C 180,E1 -10927.492,E2 -10927.492} C_VEL
LIN {X 0,Y 404.119,Z 287.771,A -85,B 0,C 180,E1 -10930.074,E2 -10930.074} C_VEL
LIN {X 0,Y 404.142,Z 287.763,A -85,B 0,C 180,E1 -10933.081,E2 -10933.081} C_VEL
LIN {X 0,Y 404.121,Z 287.77,A -85,B 0,C 180,E1 -10935.921,E2 -10935.921} C_VEL
LIN {X 0,Y 404.102,Z 287.776,A -85,B 0,C 180,E1 -10938.632,E2 -10938.632} C_VEL
LIN {X 0,Y 404.137,Z 287.765,A -85,B 0,C 180,E1 -10941.494,E2 -10941.494} C_VEL
LIN {X 0,Y 404.171,Z 287.758,A -85,B 0,C 180,E1 -10944.981,E2 -10944.981} C_VEL
LIN {X 0,Y 404.137,Z 287.767,A -85,B 0,C 180,E1 -10948.441,E2 -10948.441} C_VEL
LIN {X 0,Y 404.15,Z 287.765,A -85,B 0,C 180,E1 -10950.861,E2 -10950.861} C_VEL
LIN {X 0,Y 404.15,Z 287.767,A -85,B 0,C 180,E1 -10954.722,E2 -10954.722} C_VEL
LIN {X 0,Y 404.164,Z 287.766,A -85,B 0,C 180,E1 -10957.506,E2 -10957.506} C_VEL
LIN {X 0,Y 404.158,Z 287.762,A -85,B 0,C 180,E1 -10960.706,E2 -10960.706} C_VEL
LIN {X 0,Y 404.215,Z 287.759,A -85,B 0,C 180,E1 -10963.847,E2 -10963.847} C_VEL
LIN {X 0,Y 404.28,Z 287.729,A -85,B 0,C 180,E1 -10966.937,E2 -10966.937} C_VEL
LIN {X 0,Y 404.236,Z 287.753,A -85,B 0,C 180,E1 -10969.986,E2 -10969.986} C_VEL
LIN {X 0,Y 404.335,Z 287.742,A -85,B 0,C 180,E1 -10973.01,E2 -10973.01} C_VEL
LIN {X 0,Y 404.246,Z 287.747,A -85,B 0,C 180,E1 -10975.012,E2 -10975.012} C_VEL
LIN {X 0,Y 404.459,Z 287.715,A -85,B 0,C 180,E1 -10978.007,E2 -10978.007} C_VEL
LIN {X 0,Y 404.466,Z 287.726,A -85,B 0,C 180,E1 -10981.99,E2 -10981.99} C_VEL
LIN {X 0,Y 404.302,Z 287.72,A -85,B 0,C 180,E1 -10986.44,E2 -10986.44} C_VEL
LIN {X 0,Y 404.233,Z 287.745,A -85,B 0,C 180,E1 -10989,E2 -10989} C_VEL
LIN {X 0,Y 404.244,Z 287.753,A -85,B 0,C 180,E1 -10992.04,E2 -10992.04} C_VEL
LIN {X 0,Y 404.185,Z 287.75,A -85,B 0,C 180,E1 -10995.117,E2 -10995.117} C_VEL
LIN {X 0,Y 404.19,Z 287.744,A -85,B 0,C 180,E1 -10998.237,E2 -10998.237} C_VEL
LIN {X 0,Y 404.147,Z 287.77,A -85,B 0,C 180,E1 -11001.417,E2 -11001.417} C_VEL
LIN {X 0,Y 404.123,Z 287.763,A -85,B 0,C 180,E1 -11004.667,E2 -11004.667} C_VEL
LIN {X 0,Y 404.09,Z 287.756,A -85,B 0,C 180,E1 -11008.005,E2 -11008.005} C_VEL
LIN {X 0,Y 404.13,Z 287.763,A -85,B 0,C 180,E1 -11010.284,E2 -11010.284} C_VEL
LIN {X 0,Y 404.124,Z 287.764,A -85,B 0,C 180,E1 -11013.811,E2 -11013.811} C_VEL
LIN {X 0,Y 404.12,Z 287.75,A -85,B 0,C 180,E1 -11016.873,E2 -11016.873} C_VEL
LIN {X 0,Y 404.102,Z 287.77,A -85,B 0,C 180,E1 -11020.073,E2 -11020.073} C_VEL
LIN {X 0,Y 404.129,Z 287.766,A -85,B 0,C 180,E1 -11023.081,E2 -11023.081} C_VEL
LIN {X 0,Y 404.131,Z 287.755,A -85,B 0,C 180,E1 -11025.924,E2 -11025.924} C_VEL
LIN {X 0,Y 404.099,Z 287.773,A -85,B 0,C 180,E1 -11028.633,E2 -11028.633} C_VEL
LIN {X 0,Y 404.134,Z 287.761,A -85,B 0,C 180,E1 -11031.492,E2 -11031.492} C_VEL
LIN {X 0,Y 404.167,Z 287.763,A -85,B 0,C 180,E1 -11034.983,E2 -11034.983} C_VEL
LIN {X 0,Y 404.122,Z 287.768,A -85,B 0,C 180,E1 -11038.441,E2 -11038.441} C_VEL
LIN {X 0,Y 404.178,Z 287.761,A -85,B 0,C 180,E1 -11041.999,E2 -11041.999} C_VEL
LIN {X 0,Y 404.153,Z 287.761,A -85,B 0,C 180,E1 -11045.333,E2 -11045.333} C_VEL
LIN {X 0,Y 404.121,Z 287.771,A -85,B 0,C 180,E1 -11048.58,E2 -11048.58} C_VEL
LIN {X 0,Y 404.192,Z 287.761,A -85,B 0,C 180,E1 -11051.761,E2 -11051.761} C_VEL
LIN {X 0,Y 404.189,Z 287.765,A -85,B 0,C 180,E1 -11054.881,E2 -11054.881} C_VEL
LIN {X 0,Y 404.253,Z 287.753,A -85,B 0,C 180,E1 -11057.958,E2 -11057.958} C_VEL
LIN {X 0,Y 404.365,Z 287.738,A -85,B 0,C 180,E1 -11062.007,E2 -11062.007} C_VEL
LIN {X 0,Y 404.401,Z 287.735,A -85,B 0,C 180,E1 -11064.014,E2 -11064.014} C_VEL
LIN {X 0,Y 404.462,Z 287.725,A -85,B 0,C 180,E1 -11068.008,E2 -11068.008} C_VEL
LIN {X 0,Y 404.569,Z 287.79,A -85,B 0,C 180,E1 -11069.875,E2 -11069.875} C_VEL
LIN {X 0,Y 406.669,Z 297.231,A -85,B 0,C 180,E1 -11071.965,E2 -11071.965} C_VEL
LIN {X 0,Y 416.654,Z 321.126,A -85,B 0,C 180,E1 -11073.132,E2 -11073.132} C_VEL
LIN {X 0,Y 417.744,Z 326.6,A -85,B 0,C 180,E1 -11073.312,E2 -11073.312} C_VEL
LIN {X 0,Y 415.934,Z 416.132,A -85,B 0,C 180,E1 -11074.917,E2 -11074.917} C_VEL
LIN {X 0,Y 415.206,Z 421.984,A -85,B 0,C 180,E1 -11074.984,E2 -11074.984} C_VEL
LIN {X 0,Y 409.465,Z 441.004,A -85,B 0,C 180,E1 -11074.993,E2 -11074.993} C_VEL
LIN {X 0,Y 408.802,Z 446.851,A -85,B 0,C 180,E1 -11075.066,E2 -11075.066} C_VEL
LIN {X 0,Y 408.311,Z 466.758,A -85,B 0,C 180,E1 -11075.494,E2 -11075.494} C_VEL
LIN {X 0,Y 407.54,Z 482.278,A -85,B 0,C 180,E1 -11076.032,E2 -11076.032} C_VEL
LIN {X 0,Y 406.533,Z 497.283,A -85,B 0,C 180,E1 -11076.763,E2 -11076.763} C_VEL
LIN {X 0,Y 405.512,Z 510.39,A -85,B 0,C 180,E1 -11077.593,E2 -11077.593} C_VEL
LIN {X 0,Y 404.231,Z 523.899,A -85,B 0,C 180,E1 -11078.653,E2 -11078.653} C_VEL
LIN {X 0,Y 402.852,Z 537.033,A -85,B 0,C 180,E1 -11079.92,E2 -11079.92} C_VEL
LIN {X 0,Y 401.447,Z 549.5,A -85,B 0,C 180,E1 -11081.384,E2 -11081.384} C_VEL
LIN {X 0,Y 400.194,Z 560.469,A -85,B 0,C 180,E1 -11082.938,E2 -11082.938} C_VEL
LIN {X 0,Y 399.054,Z 569.954,A -85,B 0,C 180,E1 -11084.536,E2 -11084.536} C_VEL
LIN {X 0,Y 397.958,Z 579.205,A -85,B 0,C 180,E1 -11086.412,E2 -11086.412} C_VEL
LIN {X 0,Y 397.279,Z 585.883,A -85,B 0,C 180,E1 -11088.033,E2 -11088.033} C_VEL
LIN {X 0,Y 396.615,Z 592.831,A -85,B 0,C 180,E1 -11090.097,E2 -11090.097} C_VEL
LIN {X 0,Y 396.261,Z 597.539,A -85,B 0,C 180,E1 -11091.866,E2 -11091.866} C_VEL
LIN {X 0,Y 396.026,Z 601.107,A -85,B 0,C 180,E1 -11093.533,E2 -11093.533} C_VEL
LIN {X 0,Y 395.712,Z 603.842,A -85,B 0,C 180,E1 -11095.229,E2 -11095.229} C_VEL
LIN {X 0,Y 395.568,Z 606.239,A -85,B 0,C 180,E1 -11097.511,E2 -11097.511} C_VEL
LIN {X 0,Y 395.494,Z 607.197,A -85,B 0,C 180,E1 -11099.838,E2 -11099.838} C_VEL
LIN {X 0,Y 395.557,Z 606.977,A -85,B 0,C 180,E1 -11101.484,E2 -11101.484} C_VEL
LIN {X 0,Y 395.635,Z 605.781,A -85,B 0,C 180,E1 -11103.412,E2 -11103.412} C_VEL
LIN {X 0,Y 395.803,Z 603.648,A -85,B 0,C 180,E1 -11105.24,E2 -11105.24} C_VEL
LIN {X 0,Y 396.11,Z 600.523,A -85,B 0,C 180,E1 -11107.101,E2 -11107.101} C_VEL
LIN {X 0,Y 396.487,Z 595.88,A -85,B 0,C 180,E1 -11109.146,E2 -11109.146} C_VEL
LIN {X 0,Y 396.962,Z 590.695,A -85,B 0,C 180,E1 -11110.923,E2 -11110.923} C_VEL
LIN {X 0,Y 397.73,Z 583.706,A -85,B 0,C 180,E1 -11112.866,E2 -11112.866} C_VEL
LIN {X 0,Y 398.71,Z 575.016,A -85,B 0,C 180,E1 -11114.834,E2 -11114.834} C_VEL
LIN {X 0,Y 399.827,Z 566.433,A -85,B 0,C 180,E1 -11116.441,E2 -11116.441} C_VEL
LIN {X 0,Y 401.083,Z 556.163,A -85,B 0,C 180,E1 -11118.064,E2 -11118.064} C_VEL
LIN {X 0,Y 402.518,Z 544.804,A -85,B 0,C 180,E1 -11119.557,E2 -11119.557} C_VEL
LIN {X 0,Y 403.959,Z 532.258,A -85,B 0,C 180,E1 -11120.928,E2 -11120.928} C_VEL
LIN {X 0,Y 405.448,Z 518.396,A -85,B 0,C 180,E1 -11122.162,E2 -11122.162} C_VEL
LIN {X 0,Y 406.735,Z 504.581,A -85,B 0,C 180,E1 -11123.15,E2 -11123.15} C_VEL
LIN {X 0,Y 407.87,Z 489.845,A -85,B 0,C 180,E1 -11123.974,E2 -11123.974} C_VEL
LIN {X 0,Y 408.76,Z 475.003,A -85,B 0,C 180,E1 -11124.592,E2 -11124.592} C_VEL
LIN {X 0,Y 409.412,Z 459.689,A -85,B 0,C 180,E1 -11125.023,E2 -11125.023} C_VEL
LIN {X 0,Y 412.365,Z 327.564,A -85,B 0,C 180,E1 -11127.479,E2 -11127.479} C_VEL
LIN {X 0,Y 411.14,Z 323.447,A -85,B 0,C 180,E1 -11127.659,E2 -11127.659} C_VEL
LIN {X 0,Y 402.966,Z 305.223,A -85,B 0,C 180,E1 -11128.703,E2 -11128.703} C_VEL
LIN {X 0,Y 399.626,Z 298.33,A -85,B 0,C 180,E1 -11129.14,E2 -11129.14} C_VEL
LIN {X 0,Y 397.151,Z 288.638,A -85,B 0,C 180,E1 -11131.52,E2 -11131.52} C_VEL
LIN {X 0,Y 397.141,Z 288.64,A -85,B 0,C 180,E1 -11134.87,E2 -11134.87} C_VEL
LIN {X 0,Y 397.082,Z 288.647,A -85,B 0,C 180,E1 -11138.183,E2 -11138.183} C_VEL
LIN {X 0,Y 397.147,Z 288.638,A -85,B 0,C 180,E1 -11141.428,E2 -11141.428} C_VEL
LIN {X 0,Y 397.165,Z 288.639,A -85,B 0,C 180,E1 -11144.609,E2 -11144.609} C_VEL
LIN {X 0,Y 397.205,Z 288.633,A -85,B 0,C 180,E1 -11147.743,E2 -11147.743} C_VEL
LIN {X 0,Y 397.24,Z 288.63,A -85,B 0,C 180,E1 -11150.84,E2 -11150.84} C_VEL
LIN {X 0,Y 397.359,Z 288.608,A -85,B 0,C 180,E1 -11153.91,E2 -11153.91} C_VEL
LIN {X 0,Y 397.437,Z 288.602,A -85,B 0,C 180,E1 -11157.975,E2 -11157.975} C_VEL
LIN {X 0,Y 397.568,Z 288.585,A -85,B 0,C 180,E1 -11160.002,E2 -11160.002} C_VEL
LIN {X 0,Y 397.36,Z 288.615,A -85,B 0,C 180,E1 -11163.043,E2 -11163.043} C_VEL
LIN {X 0,Y 397.321,Z 288.615,A -85,B 0,C 180,E1 -11167.114,E2 -11167.114} C_VEL
LIN {X 0,Y 397.206,Z 288.632,A -85,B 0,C 180,E1 -11170.193,E2 -11170.193} C_VEL
LIN {X 0,Y 397.219,Z 288.627,A -85,B 0,C 180,E1 -11173.323,E2 -11173.323} C_VEL
LIN {X 0,Y 397.174,Z 288.632,A -85,B 0,C 180,E1 -11177.157,E2 -11177.157} C_VEL
LIN {X 0,Y 397.095,Z 288.645,A -85,B 0,C 180,E1 -11180.732,E2 -11180.732} C_VEL
LIN {X 0,Y 397.099,Z 288.643,A -85,B 0,C 180,E1 -11184.022,E2 -11184.022} C_VEL
LIN {X 0,Y 397.082,Z 288.645,A -85,B 0,C 180,E1 -11187.4,E2 -11187.4} C_VEL
LIN {X 0,Y 397.092,Z 288.643,A -85,B 0,C 180,E1 -11189.864,E2 -11189.864} C_VEL
LIN {X 0,Y 397.106,Z 288.641,A -85,B 0,C 180,E1 -11193.275,E2 -11193.275} C_VEL
LIN {X 0,Y 397.088,Z 288.643,A -85,B 0,C 180,E1 -11196.997,E2 -11196.997} C_VEL
LIN {X 0,Y 397.051,Z 288.652,A -85,B 0,C 180,E1 -11200.439,E2 -11200.439} C_VEL
LIN {X 0,Y 397.083,Z 288.646,A -85,B 0,C 180,E1 -11203.652,E2 -11203.652} C_VEL
LIN {X 0,Y 397.088,Z 288.649,A -85,B 0,C 180,E1 -11206.524,E2 -11206.524} C_VEL
LIN {X 0,Y 397.084,Z 288.649,A -85,B 0,C 180,E1 -11210.421,E2 -11210.421} C_VEL
LIN {X 0,Y 397.091,Z 288.64,A -85,B 0,C 180,E1 -11213.006,E2 -11213.006} C_VEL
LIN {X 0,Y 397.156,Z 288.808,A -85,B 0,C 180,E1 -11215.242,E2 -11215.242} C_VEL
LIN {X 0,Y 401.11,Z 303.469,A -85,B 0,C 180,E1 -11218.518,E2 -11218.518} C_VEL
LIN {X 0,Y 403.89,Z 315.74,A -85,B 0,C 180,E1 -11221.064,E2 -11221.064} C_VEL
LIN {X 0,Y 404.125,Z 316.755,A -85,B 0,C 180,E1 -11221.269,E2 -11221.269} C_VEL
LIN {X 0,Y 405.706,Z 321.874,A -85,B 0,C 180,E1 -11221.512,E2 -11221.512} C_VEL
LIN {X 0,Y 410.925,Z 348.189,A -85,B 0,C 180,E1 -11222.468,E2 -11222.468} C_VEL
LIN {X 0,Y 411.943,Z 355.177,A -85,B 0,C 180,E1 -11222.688,E2 -11222.688} C_VEL
LIN {X 0,Y 408.988,Z 483.493,A -85,B 0,C 180,E1 -11225.069,E2 -11225.069} C_VEL
LIN {X 0,Y 408.141,Z 499.39,A -85,B 0,C 180,E1 -11225.557,E2 -11225.557} C_VEL
LIN {X 0,Y 407.094,Z 514.048,A -85,B 0,C 180,E1 -11226.205,E2 -11226.205} C_VEL
LIN {X 0,Y 405.779,Z 528.748,A -85,B 0,C 180,E1 -11227.065,E2 -11227.065} C_VEL
LIN {X 0,Y 404.45,Z 542.144,A -85,B 0,C 180,E1 -11228.063,E2 -11228.063} C_VEL
LIN {X 0,Y 402.877,Z 555.814,A -85,B 0,C 180,E1 -11229.315,E2 -11229.315} C_VEL
LIN {X 0,Y 401.44,Z 568.321,A -85,B 0,C 180,E1 -11230.717,E2 -11230.717} C_VEL
LIN {X 0,Y 400.216,Z 578.651,A -85,B 0,C 180,E1 -11232.104,E2 -11232.104} C_VEL
LIN {X 0,Y 398.958,Z 588.338,A -85,B 0,C 180,E1 -11233.63,E2 -11233.63} C_VEL
LIN {X 0,Y 397.888,Z 597.877,A -85,B 0,C 180,E1 -11235.423,E2 -11235.423} C_VEL
LIN {X 0,Y 397.122,Z 605.833,A -85,B 0,C 180,E1 -11237.22,E2 -11237.22} C_VEL
LIN {X 0,Y 396.446,Z 613.265,A -85,B 0,C 180,E1 -11239.273,E2 -11239.273} C_VEL
LIN {X 0,Y 396.061,Z 619.165,A -85,B 0,C 180,E1 -11241.326,E2 -11241.326} C_VEL
LIN {X 0,Y 395.841,Z 622.679,A -85,B 0,C 180,E1 -11242.861,E2 -11242.861} C_VEL
LIN {X 0,Y 395.739,Z 626.22,A -85,B 0,C 180,E1 -11244.906,E2 -11244.906} C_VEL
LIN {X 0,Y 395.707,Z 628.543,A -85,B 0,C 180,E1 -11246.946,E2 -11246.946} C_VEL
LIN {X 0,Y 395.79,Z 629.701,A -85,B 0,C 180,E1 -11248.983,E2 -11248.983} C_VEL
LIN {X 0,Y 395.791,Z 629.695,A -85,B 0,C 180,E1 -11251.018,E2 -11251.018} C_VEL
LIN {X 0,Y 395.708,Z 628.474,A -85,B 0,C 180,E1 -11253.055,E2 -11253.055} C_VEL
LIN {X 0,Y 395.754,Z 626.083,A -85,B 0,C 180,E1 -11255.094,E2 -11255.094} C_VEL
LIN {X 0,Y 395.897,Z 622.468,A -85,B 0,C 180,E1 -11257.139,E2 -11257.139} C_VEL
LIN {X 0,Y 396.1,Z 617.533,A -85,B 0,C 180,E1 -11259.189,E2 -11259.189} C_VEL
LIN {X 0,Y 396.598,Z 611.153,A -85,B 0,C 180,E1 -11261.241,E2 -11261.241} C_VEL
LIN {X 0,Y 397.195,Z 603.139,A -85,B 0,C 180,E1 -11263.299,E2 -11263.299} C_VEL
LIN {X 0,Y 398.148,Z 594.605,A -85,B 0,C 180,E1 -11265.092,E2 -11265.092} C_VEL
LIN {X 0,Y 399.031,Z 585.942,A -85,B 0,C 180,E1 -11266.631,E2 -11266.631} C_VEL
LIN {X 0,Y 400.328,Z 575.685,A -85,B 0,C 180,E1 -11268.156,E2 -11268.156} C_VEL
LIN {X 0,Y 401.702,Z 563.482,A -85,B 0,C 180,E1 -11269.681,E2 -11269.681} C_VEL
LIN {X 0,Y 403.03,Z 551.244,A -85,B 0,C 180,E1 -11270.945,E2 -11270.945} C_VEL
LIN {X 0,Y 404.425,Z 537.949,A -85,B 0,C 180,E1 -11272.073,E2 -11272.073} C_VEL
LIN {X 0,Y 405.587,Z 525.301,A -85,B 0,C 180,E1 -11272.947,E2 -11272.947} C_VEL
LIN {X 0,Y 406.741,Z 510.007,A -85,B 0,C 180,E1 -11273.781,E2 -11273.781} C_VEL
LIN {X 0,Y 407.699,Z 495.369,A -85,B 0,C 180,E1 -11274.364,E2 -11274.364} C_VEL
LIN {X 0,Y 408.362,Z 480.431,A -85,B 0,C 180,E1 -11274.769,E2 -11274.769} C_VEL
LIN {X 0,Y 410.986,Z 353.594,A -85,B 0,C 180,E1 -11277.09,E2 -11277.09} C_VEL
LIN {X 0,Y 404.197,Z 318.753,A -85,B 0,C 180,E1 -11278.258,E2 -11278.258} C_VEL
LIN {X 0,Y 403.966,Z 317.414,A -85,B 0,C 180,E1 -11278.342,E2 -11278.342} C_VEL
LIN {X 0,Y 401.635,Z 306.495,A -85,B 0,C 180,E1 -11280.494,E2 -11280.494} C_VEL
LIN {X 0,Y 398.405,Z 293.682,A -85,B 0,C 180,E1 -11283.151,E2 -11283.151} C_VEL
LIN {X 0,Y 397.117,Z 288.645,A -85,B 0,C 180,E1 -11284.28,E2 -11284.28} C_VEL
LIN {X 0,Y 397.09,Z 288.651,A -85,B 0,C 180,E1 -11287.207,E2 -11287.207} C_VEL
LIN {X 0,Y 397.056,Z 288.648,A -85,B 0,C 180,E1 -11290.436,E2 -11290.436} C_VEL
LIN {X 0,Y 397.087,Z 288.642,A -85,B 0,C 180,E1 -11293.65,E2 -11293.65} C_VEL
LIN {X 0,Y 397.092,Z 288.642,A -85,B 0,C 180,E1 -11296.522,E2 -11296.522} C_VEL
LIN {X 0,Y 397.086,Z 288.642,A -85,B 0,C 180,E1 -11300.418,E2 -11300.418} C_VEL
LIN {X 0,Y 397.092,Z 288.648,A -85,B 0,C 180,E1 -11303.003,E2 -11303.003} C_VEL
LIN {X 0,Y 397.111,Z 288.639,A -85,B 0,C 180,E1 -11306.725,E2 -11306.725} C_VEL
LIN {X 0,Y 397.116,Z 288.644,A -85,B 0,C 180,E1 -11310.294,E2 -11310.294} C_VEL
LIN {X 0,Y 397.073,Z 288.649,A -85,B 0,C 180,E1 -11313.736,E2 -11313.736} C_VEL
LIN {X 0,Y 397.097,Z 288.643,A -85,B 0,C 180,E1 -11317.084,E2 -11317.084} C_VEL
LIN {X 0,Y 397.143,Z 288.637,A -85,B 0,C 180,E1 -11320.351,E2 -11320.351} C_VEL
LIN {X 0,Y 397.162,Z 288.642,A -85,B 0,C 180,E1 -11323.552,E2 -11323.552} C_VEL
LIN {X 0,Y 397.226,Z 288.608,A -85,B 0,C 180,E1 -11326.701,E2 -11326.701} C_VEL
LIN {X 0,Y 397.198,Z 288.626,A -85,B 0,C 180,E1 -11329.807,E2 -11329.807} C_VEL
LIN {X 0,Y 397.287,Z 288.62,A -85,B 0,C 180,E1 -11332.885,E2 -11332.885} C_VEL
LIN {X 0,Y 397.218,Z 288.622,A -85,B 0,C 180,E1 -11334.923,E2 -11334.923} C_VEL
LIN {X 0,Y 397.427,Z 288.589,A -85,B 0,C 180,E1 -11337.972,E2 -11337.972} C_VEL
LIN {X 0,Y 397.434,Z 288.602,A -85,B 0,C 180,E1 -11342.025,E2 -11342.025} C_VEL
LIN {X 0,Y 397.26,Z 288.596,A -85,B 0,C 180,E1 -11346.433,E2 -11346.433} C_VEL
LIN {X 0,Y 397.183,Z 288.624,A -85,B 0,C 180,E1 -11349.162,E2 -11349.162} C_VEL
LIN {X 0,Y 397.208,Z 288.629,A -85,B 0,C 180,E1 -11352.257,E2 -11352.257} C_VEL
LIN {X 0,Y 397.16,Z 288.62,A -85,B 0,C 180,E1 -11355.391,E2 -11355.391} C_VEL
LIN {X 0,Y 397.145,Z 288.622,A -85,B 0,C 180,E1 -11358.572,E2 -11358.572} C_VEL
LIN {X 0,Y 397.095,Z 288.645,A -85,B 0,C 180,E1 -11361.816,E2 -11361.816} C_VEL
LIN {X 0,Y 397.091,Z 288.634,A -85,B 0,C 180,E1 -11365.134,E2 -11365.134} C_VEL
LIN {X 0,Y 397.05,Z 288.633,A -85,B 0,C 180,E1 -11368.547,E2 -11368.547} C_VEL
LIN {X 0,Y 397.067,Z 288.648,A -85,B 0,C 180,E1 -11371.834,E2 -11371.834} C_VEL
LIN {X 0,Y 397.103,Z 288.638,A -85,B 0,C 180,E1 -11374.493,E2 -11374.493} C_VEL
LIN {X 0,Y 397.078,Z 288.635,A -85,B 0,C 180,E1 -11378.275,E2 -11378.275} C_VEL
LIN {X 0,Y 397.038,Z 288.65,A -85,B 0,C 180,E1 -11381.975,E2 -11381.975} C_VEL
LIN {X 0,Y 397.069,Z 288.633,A -85,B 0,C 180,E1 -11385.068,E2 -11385.068} C_VEL
LIN {X 0,Y 397.046,Z 288.649,A -85,B 0,C 180,E1 -11388.021,E2 -11388.021} C_VEL
LIN {X 0,Y 397.11,Z 288.64,A -85,B 0,C 180,E1 -11391.138,E2 -11391.138} C_VEL
LIN {X 0,Y 397.102,Z 288.637,A -85,B 0,C 180,E1 -11394.496,E2 -11394.496} C_VEL
LIN {X 0,Y 397.061,Z 288.646,A -85,B 0,C 180,E1 -11397.927,E2 -11397.927} C_VEL
LIN {X 0,Y 397.1,Z 288.644,A -85,B 0,C 180,E1 -11401.455,E2 -11401.455} C_VEL
LIN {X 0,Y 397.135,Z 288.635,A -85,B 0,C 180,E1 -11404.487,E2 -11404.487} C_VEL
LIN {X 0,Y 397.078,Z 288.648,A -85,B 0,C 180,E1 -11408.181,E2 -11408.181} C_VEL
LIN {X 0,Y 397.144,Z 288.64,A -85,B 0,C 180,E1 -11411.426,E2 -11411.426} C_VEL
LIN {X 0,Y 397.162,Z 288.637,A -85,B 0,C 180,E1 -11414.607,E2 -11414.607} C_VEL
LIN {X 0,Y 397.212,Z 288.63,A -85,B 0,C 180,E1 -11417.742,E2 -11417.742} C_VEL
LIN {X 0,Y 397.241,Z 288.63,A -85,B 0,C 180,E1 -11420.838,E2 -11420.838} C_VEL
LIN {X 0,Y 397.352,Z 288.613,A -85,B 0,C 180,E1 -11423.908,E2 -11423.908} C_VEL
LIN {X 0,Y 397.431,Z 288.601,A -85,B 0,C 180,E1 -11427.973,E2 -11427.973} C_VEL
LIN {X 0,Y 397.457,Z 288.702,A -85,B 0,C 180,E1 -11429.461,E2 -11429.461} C_VEL
LIN {X 0,Y 399.471,Z 297.323,A -85,B 0,C 180,E1 -11431.434,E2 -11431.434} C_VEL
LIN {X 0,Y 410.514,Z 323.409,A -85,B 0,C 180,E1 -11432.758,E2 -11432.758} C_VEL
LIN {X 0,Y 411.347,Z 327.877,A -85,B 0,C 180,E1 -11432.904,E2 -11432.904} C_VEL
LIN {X 0,Y 408.802,Z 446.851,A -85,B 0,C 180,E1 -11435.066,E2 -11435.066} C_VEL
LIN {X 0,Y 408.151,Z 452.688,A -85,B 0,C 180,E1 -11435.137,E2 -11435.137} C_VEL
LIN {X 0,Y 405.324,Z 462.179,A -85,B 0,C 180,E1 -11435.174,E2 -11435.174} C_VEL
LIN {X 0,Y 402.325,Z 471.602,A -85,B 0,C 180,E1 -11435.28,E2 -11435.28} C_VEL
LIN {X 0,Y 401.357,Z 477.334,A -85,B 0,C 180,E1 -11435.438,E2 -11435.438} C_VEL
LIN {X 0,Y 400.387,Z 492.421,A -85,B 0,C 180,E1 -11436.108,E2 -11436.108} C_VEL
LIN {X 0,Y 399.241,Z 506.648,A -85,B 0,C 180,E1 -11436.951,E2 -11436.951} C_VEL
LIN {X 0,Y 397.954,Z 520.539,A -85,B 0,C 180,E1 -11437.994,E2 -11437.994} C_VEL
LIN {X 0,Y 396.546,Z 533.36,A -85,B 0,C 180,E1 -11439.178,E2 -11439.178} C_VEL
LIN {X 0,Y 395.211,Z 545.183,A -85,B 0,C 180,E1 -11440.502,E2 -11440.502} C_VEL
LIN {X 0,Y 393.937,Z 555.881,A -85,B 0,C 180,E1 -11441.93,E2 -11441.93} C_VEL
LIN {X 0,Y 392.727,Z 565.534,A -85,B 0,C 180,E1 -11443.452,E2 -11443.452} C_VEL
LIN {X 0,Y 391.643,Z 574.284,A -85,B 0,C 180,E1 -11445.081,E2 -11445.081} C_VEL
LIN {X 0,Y 390.793,Z 581.695,A -85,B 0,C 180,E1 -11446.722,E2 -11446.722} C_VEL
LIN {X 0,Y 390.086,Z 587.987,A -85,B 0,C 180,E1 -11448.377,E2 -11448.377} C_VEL
LIN {X 0,Y 389.489,Z 593.883,A -85,B 0,C 180,E1 -11450.241,E2 -11450.241} C_VEL
LIN {X 0,Y 389.113,Z 599.015,A -85,B 0,C 180,E1 -11452.289,E2 -11452.289} C_VEL
LIN {X 0,Y 388.96,Z 601.288,A -85,B 0,C 180,E1 -11453.422,E2 -11453.422} C_VEL
LIN {X 0,Y 388.583,Z 604.776,A -85,B 0,C 180,E1 -11455.725,E2 -11455.725} C_VEL
LIN {X 0,Y 388.478,Z 606.513,A -85,B 0,C 180,E1 -11457.574,E2 -11457.574} C_VEL
LIN {X 0,Y 388.393,Z 607.378,A -85,B 0,C 180,E1 -11459.713,E2 -11459.713} C_VEL
LIN {X 0,Y 388.459,Z 607.078,A -85,B 0,C 180,E1 -11461.758,E2 -11461.758} C_VEL
LIN {X 0,Y 388.576,Z 605.372,A -85,B 0,C 180,E1 -11464.102,E2 -11464.102} C_VEL
LIN {X 0,Y 388.747,Z 603.562,A -85,B 0,C 180,E1 -11465.561,E2 -11465.561} C_VEL
LIN {X 0,Y 389.154,Z 599.444,A -85,B 0,C 180,E1 -11467.88,E2 -11467.88} C_VEL
LIN {X 0,Y 389.578,Z 594.748,A -85,B 0,C 180,E1 -11469.822,E2 -11469.822} C_VEL
LIN {X 0,Y 390.215,Z 588.756,A -85,B 0,C 180,E1 -11471.788,E2 -11471.788} C_VEL
LIN {X 0,Y 391.127,Z 580.969,A -85,B 0,C 180,E1 -11473.84,E2 -11473.84} C_VEL
LIN {X 0,Y 392.294,Z 571.952,A -85,B 0,C 180,E1 -11475.773,E2 -11475.773} C_VEL
LIN {X 0,Y 393.652,Z 561.39,A -85,B 0,C 180,E1 -11477.635,E2 -11477.635} C_VEL
LIN {X 0,Y 395.141,Z 550.341,A -85,B 0,C 180,E1 -11479.241,E2 -11479.241} C_VEL
LIN {X 0,Y 396.619,Z 538.502,A -85,B 0,C 180,E1 -11480.675,E2 -11480.675} C_VEL
LIN {X 0,Y 398.148,Z 525.599,A -85,B 0,C 180,E1 -11481.964,E2 -11481.964} C_VEL
LIN {X 0,Y 399.587,Z 511.918,A -85,B 0,C 180,E1 -11483.076,E2 -11483.076} C_VEL
LIN {X 0,Y 400.836,Z 498.204,A -85,B 0,C 180,E1 -11483.967,E2 -11483.967} C_VEL
LIN {X 0,Y 401.887,Z 483.548,A -85,B 0,C 180,E1 -11484.703,E2 -11484.703} C_VEL
LIN {X 0,Y 402.729,Z 468.654,A -85,B 0,C 180,E1 -11485.242,E2 -11485.242} C_VEL
LIN {X 0,Y 403.258,Z 451.938,A -85,B 0,C 180,E1 -11485.63,E2 -11485.63} C_VEL
LIN {X 0,Y 406.127,Z 328.683,A -85,B 0,C 180,E1 -11487.948,E2 -11487.948} C_VEL
LIN {X 0,Y 401.243,Z 316.984,A -85,B 0,C 180,E1 -11488.597,E2 -11488.597} C_VEL
LIN {X 0,Y 393.696,Z 301.326,A -85,B 0,C 180,E1 -11489.598,E2 -11489.598} C_VEL
LIN {X 0,Y 392.446,Z 298.523,A -85,B 0,C 180,E1 -11489.789,E2 -11489.789} C_VEL
LIN {X 0,Y 390.101,Z 289.519,A -85,B 0,C 180,E1 -11492.071,E2 -11492.071} C_VEL
LIN {X 0,Y 390.064,Z 289.52,A -85,B 0,C 180,E1 -11495.521,E2 -11495.521} C_VEL
LIN {X 0,Y 390.041,Z 289.528,A -85,B 0,C 180,E1 -11498.879,E2 -11498.879} C_VEL
LIN {X 0,Y 390.114,Z 289.518,A -85,B 0,C 180,E1 -11502.168,E2 -11502.168} C_VEL
LIN {X 0,Y 390.13,Z 289.515,A -85,B 0,C 180,E1 -11505.394,E2 -11505.394} C_VEL
LIN {X 0,Y 390.134,Z 289.514,A -85,B 0,C 180,E1 -11508.573,E2 -11508.573} C_VEL
LIN {X 0,Y 390.296,Z 289.491,A -85,B 0,C 180,E1 -11512.033,E2 -11512.033} C_VEL
LIN {X 0,Y 390.212,Z 289.503,A -85,B 0,C 180,E1 -11514.835,E2 -11514.835} C_VEL
LIN {X 0,Y 390.406,Z 289.478,A -85,B 0,C 180,E1 -11517.938,E2 -11517.938} C_VEL
LIN {X 0,Y 390.538,Z 289.46,A -85,B 0,C 180,E1 -11520.002,E2 -11520.002} C_VEL
LIN {X 0,Y 390.294,Z 289.496,A -85,B 0,C 180,E1 -11523.098,E2 -11523.098} C_VEL
LIN {X 0,Y 390.294,Z 289.492,A -85,B 0,C 180,E1 -11526.204,E2 -11526.204} C_VEL
LIN {X 0,Y 390.183,Z 289.507,A -85,B 0,C 180,E1 -11529.331,E2 -11529.331} C_VEL
LIN {X 0,Y 390.161,Z 289.511,A -85,B 0,C 180,E1 -11532.485,E2 -11532.485} C_VEL
LIN {X 0,Y 390.13,Z 289.512,A -85,B 0,C 180,E1 -11535.679,E2 -11535.679} C_VEL
LIN {X 0,Y 390.095,Z 289.518,A -85,B 0,C 180,E1 -11538.924,E2 -11538.924} C_VEL
LIN {X 0,Y 390.028,Z 289.528,A -85,B 0,C 180,E1 -11542.236,E2 -11542.236} C_VEL
LIN {X 0,Y 390.044,Z 289.521,A -85,B 0,C 180,E1 -11545.724,E2 -11545.724} C_VEL
LIN {X 0,Y 390.022,Z 289.523,A -85,B 0,C 180,E1 -11549.114,E2 -11549.114} C_VEL
LIN {X 0,Y 390.035,Z 289.525,A -85,B 0,C 180,E1 -11552.724,E2 -11552.724} C_VEL
LIN {X 0,Y 390.036,Z 289.525,A -85,B 0,C 180,E1 -11555.824,E2 -11555.824} C_VEL
LIN {X 0,Y 390.031,Z 289.52,A -85,B 0,C 180,E1 -11559.213,E2 -11559.213} C_VEL
LIN {X 0,Y 390.026,Z 289.529,A -85,B 0,C 180,E1 -11562.373,E2 -11562.373} C_VEL
LIN {X 0,Y 390.037,Z 289.525,A -85,B 0,C 180,E1 -11565.355,E2 -11565.355} C_VEL
LIN {X 0,Y 390.012,Z 289.531,A -85,B 0,C 180,E1 -11568.186,E2 -11568.186} C_VEL
LIN {X 0,Y 390.054,Z 289.524,A -85,B 0,C 180,E1 -11570.905,E2 -11570.905} C_VEL
LIN {X 0,Y 390.115,Z 289.68,A -85,B 0,C 180,E1 -11574.683,E2 -11574.683} C_VEL
LIN {X 0,Y 393.05,Z 300.424,A -85,B 0,C 180,E1 -11577.183,E2 -11577.183} C_VEL
LIN {X 0,Y 395.819,Z 311.462,A -85,B 0,C 180,E1 -11579.601,E2 -11579.601} C_VEL
LIN {X 0,Y 396.985,Z 316.728,A -85,B 0,C 180,E1 -11580.669,E2 -11580.669} C_VEL
LIN {X 0,Y 399.611,Z 323.575,A -85,B 0,C 180,E1 -11581.043,E2 -11581.043} C_VEL
LIN {X 0,Y 404.437,Z 347.931,A -85,B 0,C 180,E1 -11581.956,E2 -11581.956} C_VEL
LIN {X 0,Y 405.713,Z 355.675,A -85,B 0,C 180,E1 -11582.218,E2 -11582.218} C_VEL
LIN {X 0,Y 402.6,Z 483.996,A -85,B 0,C 180,E1 -11584.646,E2 -11584.646} C_VEL
LIN {X 0,Y 401.698,Z 499.608,A -85,B 0,C 180,E1 -11585.138,E2 -11585.138} C_VEL
LIN {X 0,Y 400.631,Z 514.057,A -85,B 0,C 180,E1 -11585.792,E2 -11585.792} C_VEL
LIN {X 0,Y 399.244,Z 528.763,A -85,B 0,C 180,E1 -11586.668,E2 -11586.668} C_VEL
LIN {X 0,Y 397.854,Z 542.128,A -85,B 0,C 180,E1 -11587.68,E2 -11587.68} C_VEL
LIN {X 0,Y 396.208,Z 555.759,A -85,B 0,C 180,E1 -11588.95,E2 -11588.95} C_VEL
LIN {X 0,Y 394.659,Z 568.419,A -85,B 0,C 180,E1 -11590.396,E2 -11590.396} C_VEL
LIN {X 0,Y 393.391,Z 578.555,A -85,B 0,C 180,E1 -11591.782,E2 -11591.782} C_VEL
LIN {X 0,Y 392.078,Z 588.224,A -85,B 0,C 180,E1 -11593.334,E2 -11593.334} C_VEL
LIN {X 0,Y 390.941,Z 597.74,A -85,B 0,C 180,E1 -11595.158,E2 -11595.158} C_VEL
LIN {X 0,Y 390.093,Z 605.842,A -85,B 0,C 180,E1 -11597.029,E2 -11597.029} C_VEL
LIN {X 0,Y 389.414,Z 613.096,A -85,B 0,C 180,E1 -11599.077,E2 -11599.077} C_VEL
LIN {X 0,Y 388.972,Z 618.988,A -85,B 0,C 180,E1 -11601.166,E2 -11601.166} C_VEL
LIN {X 0,Y 388.784,Z 622.501,A -85,B 0,C 180,E1 -11602.731,E2 -11602.731} C_VEL
LIN {X 0,Y 388.643,Z 626.034,A -85,B 0,C 180,E1 -11604.813,E2 -11604.813} C_VEL
LIN {X 0,Y 388.613,Z 628.349,A -85,B 0,C 180,E1 -11606.89,E2 -11606.89} C_VEL
LIN {X 0,Y 388.702,Z 629.499,A -85,B 0,C 180,E1 -11608.964,E2 -11608.964} C_VEL
LIN {X 0,Y 388.703,Z 629.487,A -85,B 0,C 180,E1 -11611.036,E2 -11611.036} C_VEL
LIN {X 0,Y 388.614,Z 628.258,A -85,B 0,C 180,E1 -11613.11,E2 -11613.11} C_VEL
LIN {X 0,Y 388.66,Z 625.855,A -85,B 0,C 180,E1 -11615.188,E2 -11615.188} C_VEL
LIN {X 0,Y 388.817,Z 622.227,A -85,B 0,C 180,E1 -11617.269,E2 -11617.269} C_VEL
LIN {X 0,Y 389.032,Z 617.277,A -85,B 0,C 180,E1 -11619.357,E2 -11619.357} C_VEL
LIN {X 0,Y 389.573,Z 610.881,A -85,B 0,C 180,E1 -11621.446,E2 -11621.446} C_VEL
LIN {X 0,Y 390.222,Z 602.848,A -85,B 0,C 180,E1 -11623.541,E2 -11623.541} C_VEL
LIN {X 0,Y 391.215,Z 594.293,A -85,B 0,C 180,E1 -11625.366,E2 -11625.366} C_VEL
LIN {X 0,Y 392.153,Z 585.612,A -85,B 0,C 180,E1 -11626.931,E2 -11626.931} C_VEL
LIN {X 0,Y 393.502,Z 575.334,A -85,B 0,C 180,E1 -11628.483,E2 -11628.483} C_VEL
LIN {X 0,Y 394.929,Z 563.098,A -85,B 0,C 180,E1 -11630.033,E2 -11630.033} C_VEL
LIN {X 0,Y 396.339,Z 550.821,A -85,B 0,C 180,E1 -11631.316,E2 -11631.316} C_VEL
LIN {X 0,Y 397.797,Z 537.463,A -85,B 0,C 180,E1 -11632.461,E2 -11632.461} C_VEL
LIN {X 0,Y 399.132,Z 523.419,A -85,B 0,C 180,E1 -11633.43,E2 -11633.43} C_VEL
LIN {X 0,Y 400.207,Z 509.308,A -85,B 0,C 180,E1 -11634.194,E2 -11634.194} C_VEL
LIN {X 0,Y 401.211,Z 494.461,A -85,B 0,C 180,E1 -11634.784,E2 -11634.784} C_VEL
LIN {X 0,Y 401.881,Z 479.072,A -85,B 0,C 180,E1 -11635.196,E2 -11635.196} C_VEL
LIN {X 0,Y 404.551,Z 354.57,A -85,B 0,C 180,E1 -11637.51,E2 -11637.51} C_VEL
LIN {X 0,Y 397.904,Z 320.197,A -85,B 0,C 180,E1 -11638.686,E2 -11638.686} C_VEL
LIN {X 0,Y 396.854,Z 317.288,A -85,B 0,C 180,E1 -11638.854,E2 -11638.854} C_VEL
LIN {X 0,Y 393.925,Z 304.505,A -85,B 0,C 180,E1 -11641.455,E2 -11641.455} C_VEL
LIN {X 0,Y 390.091,Z 289.523,A -85,B 0,C 180,E1 -11644.704,E2 -11644.704} C_VEL
LIN {X 0,Y 390.038,Z 289.526,A -85,B 0,C 180,E1 -11647.78,E2 -11647.78} C_VEL
LIN {X 0,Y 390.018,Z 289.525,A -85,B 0,C 180,E1 -11650.813,E2 -11650.813} C_VEL
LIN {X 0,Y 390.044,Z 289.52,A -85,B 0,C 180,E1 -11653.883,E2 -11653.883} C_VEL
LIN {X 0,Y 390.048,Z 289.52,A -85,B 0,C 180,E1 -11656.787,E2 -11656.787} C_VEL
LIN {X 0,Y 390.01,Z 289.532,A -85,B 0,C 180,E1 -11659.553,E2 -11659.553} C_VEL
LIN {X 0,Y 390.037,Z 289.529,A -85,B 0,C 180,E1 -11662.45,E2 -11662.45} C_VEL
LIN {X 0,Y 390.061,Z 289.514,A -85,B 0,C 180,E1 -11666.043,E2 -11666.043} C_VEL
LIN {X 0,Y 390.043,Z 289.524,A -85,B 0,C 180,E1 -11669.869,E2 -11669.869} C_VEL
LIN {X 0,Y 390.029,Z 289.522,A -85,B 0,C 180,E1 -11673.224,E2 -11673.224} C_VEL
LIN {X 0,Y 390.057,Z 289.52,A -85,B 0,C 180,E1 -11676.765,E2 -11676.765} C_VEL
LIN {X 0,Y 390.101,Z 289.517,A -85,B 0,C 180,E1 -11679.981,E2 -11679.981} C_VEL
LIN {X 0,Y 390.135,Z 289.516,A -85,B 0,C 180,E1 -11683.247,E2 -11683.247} C_VEL
LIN {X 0,Y 390.192,Z 289.484,A -85,B 0,C 180,E1 -11686.56,E2 -11686.56} C_VEL
LIN {X 0,Y 390.179,Z 289.502,A -85,B 0,C 180,E1 -11690.669,E2 -11690.669} C_VEL
LIN {X 0,Y 390.269,Z 289.491,A -85,B 0,C 180,E1 -11693.796,E2 -11693.796} C_VEL
LIN {X 0,Y 390.393,Z 289.464,A -85,B 0,C 180,E1 -11697.935,E2 -11697.935} C_VEL
LIN {X 0,Y 390.402,Z 289.477,A -85,B 0,C 180,E1 -11702.062,E2 -11702.062} C_VEL
LIN {X 0,Y 390.222,Z 289.472,A -85,B 0,C 180,E1 -11706.423,E2 -11706.423} C_VEL
LIN {X 0,Y 390.153,Z 289.502,A -85,B 0,C 180,E1 -11709.328,E2 -11709.328} C_VEL
LIN {X 0,Y 390.161,Z 289.507,A -85,B 0,C 180,E1 -11712.481,E2 -11712.481} C_VEL
LIN {X 0,Y 390.122,Z 289.492,A -85,B 0,C 180,E1 -11715.675,E2 -11715.675} C_VEL
LIN {X 0,Y 390.09,Z 289.502,A -85,B 0,C 180,E1 -11718.921,E2 -11718.921} C_VEL
LIN {X 0,Y 390.031,Z 289.523,A -85,B 0,C 180,E1 -11722.232,E2 -11722.232} C_VEL
LIN {X 0,Y 390.039,Z 289.505,A -85,B 0,C 180,E1 -11725.72,E2 -11725.72} C_VEL
LIN {X 0,Y 390.011,Z 289.514,A -85,B 0,C 180,E1 -11729.111,E2 -11729.111} C_VEL
LIN {X 0,Y 390.028,Z 289.526,A -85,B 0,C 180,E1 -11732.72,E2 -11732.72} C_VEL
LIN {X 0,Y 390.029,Z 289.505,A -85,B 0,C 180,E1 -11735.821,E2 -11735.821} C_VEL
LIN {X 0,Y 390.023,Z 289.522,A -85,B 0,C 180,E1 -11739.211,E2 -11739.211} C_VEL
LIN {X 0,Y 390.017,Z 289.526,A -85,B 0,C 180,E1 -11742.371,E2 -11742.371} C_VEL
LIN {X 0,Y 390.027,Z 289.509,A -85,B 0,C 180,E1 -11745.353,E2 -11745.353} C_VEL
LIN {X 0,Y 390.012,Z 289.526,A -85,B 0,C 180,E1 -11748.185,E2 -11748.185} C_VEL
LIN {X 0,Y 390.072,Z 289.52,A -85,B 0,C 180,E1 -11750.906,E2 -11750.906} C_VEL
LIN {X 0,Y 390.068,Z 289.516,A -85,B 0,C 180,E1 -11754.792,E2 -11754.792} C_VEL
LIN {X 0,Y 390.007,Z 289.524,A -85,B 0,C 180,E1 -11758.494,E2 -11758.494} C_VEL
LIN {X 0,Y 390.101,Z 289.515,A -85,B 0,C 180,E1 -11762.069,E2 -11762.069} C_VEL
LIN {X 0,Y 390.058,Z 289.518,A -85,B 0,C 180,E1 -11765.518,E2 -11765.518} C_VEL
LIN {X 0,Y 390.07,Z 289.513,A -85,B 0,C 180,E1 -11769.529,E2 -11769.529} C_VEL
LIN {X 0,Y 390.121,Z 289.509,A -85,B 0,C 180,E1 -11773.247,E2 -11773.247} C_VEL
LIN {X 0,Y 390.177,Z 289.505,A -85,B 0,C 180,E1 -11776.561,E2 -11776.561} C_VEL
LIN {X 0,Y 390.161,Z 289.504,A -85,B 0,C 180,E1 -11779.622,E2 -11779.622} C_VEL
LIN {X 0,Y 390.285,Z 289.495,A -85,B 0,C 180,E1 -11782.758,E2 -11782.758} C_VEL
LIN {X 0,Y 390.206,Z 289.507,A -85,B 0,C 180,E1 -11784.833,E2 -11784.833} C_VEL
LIN {X 0,Y 390.4,Z 289.477,A -85,B 0,C 180,E1 -11787.936,E2 -11787.936} C_VEL
LIN {X 0,Y 390.352,Z 289.598,A -85,B 0,C 180,E1 -11789.032,E2 -11789.032} C_VEL
LIN {X 0,Y 392.309,Z 297.56,A -85,B 0,C 180,E1 -11790.898,E2 -11790.898} C_VEL
LIN {X 0,Y 404.506,Z 326.293,A -85,B 0,C 180,E1 -11792.398,E2 -11792.398} C_VEL
LIN {X 0,Y 404.944,Z 329.299,A -85,B 0,C 180,E1 -11792.49,E2 -11792.49} C_VEL
LIN {X 0,Y 401.984,Z 462.987,A -85,B 0,C 180,E1 -11794.989,E2 -11794.989} C_VEL
LIN {X 0,Y 401.357,Z 477.334,A -85,B 0,C 180,E1 -11795.438,E2 -11795.438} C_VEL
LIN {X 0,Y 400.332,Z 483.025,A -85,B 0,C 180,E1 -11795.618,E2 -11795.618} C_VEL
LIN {X 0,Y 397.066,Z 492.206,A -85,B 0,C 180,E1 -11795.886,E2 -11795.886} C_VEL
LIN {X 0,Y 393.762,Z 501.19,A -85,B 0,C 180,E1 -11796.24,E2 -11796.24} C_VEL
LIN {X 0,Y 392.682,Z 506.564,A -85,B 0,C 180,E1 -11796.553,E2 -11796.553} C_VEL
LIN {X 0,Y 391.36,Z 520.238,A -85,B 0,C 180,E1 -11797.589,E2 -11797.589} C_VEL
LIN {X 0,Y 389.881,Z 533.357,A -85,B 0,C 180,E1 -11798.813,E2 -11798.813} C_VEL
LIN {X 0,Y 388.472,Z 545.226,A -85,B 0,C 180,E1 -11800.159,E2 -11800.159} C_VEL
LIN {X 0,Y 387.208,Z 555.314,A -85,B 0,C 180,E1 -11801.516,E2 -11801.516} C_VEL
LIN {X 0,Y 385.888,Z 565.631,A -85,B 0,C 180,E1 -11803.158,E2 -11803.158} C_VEL
LIN {X 0,Y 384.743,Z 574.409,A -85,B 0,C 180,E1 -11804.816,E2 -11804.816} C_VEL
LIN {X 0,Y 383.694,Z 582.978,A -85,B 0,C 180,E1 -11806.767,E2 -11806.767} C_VEL
LIN {X 0,Y 382.915,Z 590.062,A -85,B 0,C 180,E1 -11808.734,E2 -11808.734} C_VEL
LIN {X 0,Y 382.252,Z 596.549,A -85,B 0,C 180,E1 -11811.009,E2 -11811.009} C_VEL
LIN {X 0,Y 381.94,Z 601.049,A -85,B 0,C 180,E1 -11813.075,E2 -11813.075} C_VEL
LIN {X 0,Y 381.514,Z 604.8,A -85,B 0,C 180,E1 -11815.498,E2 -11815.498} C_VEL
LIN {X 0,Y 381.381,Z 606.912,A -85,B 0,C 180,E1 -11817.812,E2 -11817.812} C_VEL
LIN {X 0,Y 381.302,Z 607.623,A -85,B 0,C 180,E1 -11819.976,E2 -11819.976} C_VEL
LIN {X 0,Y 381.386,Z 607.066,A -85,B 0,C 180,E1 -11822.302,E2 -11822.302} C_VEL
LIN {X 0,Y 381.476,Z 605.776,A -85,B 0,C 180,E1 -11824.004,E2 -11824.004} C_VEL
LIN {X 0,Y 381.764,Z 603.191,A -85,B 0,C 180,E1 -11826.091,E2 -11826.091} C_VEL
LIN {X 0,Y 382.124,Z 599.411,A -85,B 0,C 180,E1 -11828.166,E2 -11828.166} C_VEL
LIN {X 0,Y 382.568,Z 594.985,A -85,B 0,C 180,E1 -11830.012,E2 -11830.012} C_VEL
LIN {X 0,Y 383.246,Z 588.998,A -85,B 0,C 180,E1 -11832.014,E2 -11832.014} C_VEL
LIN {X 0,Y 384.171,Z 581.489,A -85,B 0,C 180,E1 -11834.039,E2 -11834.039} C_VEL
LIN {X 0,Y 385.228,Z 573.702,A -85,B 0,C 180,E1 -11835.777,E2 -11835.777} C_VEL
LIN {X 0,Y 386.428,Z 564.835,A -85,B 0,C 180,E1 -11837.439,E2 -11837.439} C_VEL
LIN {X 0,Y 387.895,Z 554.464,A -85,B 0,C 180,E1 -11839.064,E2 -11839.064} C_VEL
LIN {X 0,Y 389.366,Z 543.565,A -85,B 0,C 180,E1 -11840.498,E2 -11840.498} C_VEL
LIN {X 0,Y 390.971,Z 531.242,A -85,B 0,C 180,E1 -11841.851,E2 -11841.851} C_VEL
LIN {X 0,Y 392.539,Z 517.627,A -85,B 0,C 180,E1 -11843.078,E2 -11843.078} C_VEL
LIN {X 0,Y 393.925,Z 503.957,A -85,B 0,C 180,E1 -11844.066,E2 -11844.066} C_VEL
LIN {X 0,Y 395.151,Z 489.256,A -85,B 0,C 180,E1 -11844.896,E2 -11844.896} C_VEL
LIN {X 0,Y 396.095,Z 474.345,A -85,B 0,C 180,E1 -11845.521,E2 -11845.521} C_VEL
LIN {X 0,Y 396.8,Z 458.837,A -85,B 0,C 180,E1 -11845.954,E2 -11845.954} C_VEL
LIN {X 0,Y 399.994,Z 330.457,A -85,B 0,C 180,E1 -11848.414,E2 -11848.414} C_VEL
LIN {X 0,Y 392.381,Z 313.118,A -85,B 0,C 180,E1 -11849.455,E2 -11849.455} C_VEL
LIN {X 0,Y 385.278,Z 298.776,A -85,B 0,C 180,E1 -11850.459,E2 -11850.459} C_VEL
LIN {X 0,Y 383.041,Z 290.396,A -85,B 0,C 180,E1 -11852.699,E2 -11852.699} C_VEL
LIN {X 0,Y 383.036,Z 290.395,A -85,B 0,C 180,E1 -11855.041,E2 -11855.041} C_VEL
LIN {X 0,Y 382.978,Z 290.405,A -85,B 0,C 180,E1 -11858.47,E2 -11858.47} C_VEL
LIN {X 0,Y 383.075,Z 290.394,A -85,B 0,C 180,E1 -11861.829,E2 -11861.829} C_VEL
LIN {X 0,Y 383.096,Z 290.391,A -85,B 0,C 180,E1 -11865.12,E2 -11865.12} C_VEL
LIN {X 0,Y 383.084,Z 290.391,A -85,B 0,C 180,E1 -11868.359,E2 -11868.359} C_VEL
LIN {X 0,Y 383.252,Z 290.368,A -85,B 0,C 180,E1 -11871.977,E2 -11871.977} C_VEL
LIN {X 0,Y 383.184,Z 290.378,A -85,B 0,C 180,E1 -11874.74,E2 -11874.74} C_VEL
LIN {X 0,Y 383.374,Z 290.354,A -85,B 0,C 180,E1 -11877.901,E2 -11877.901} C_VEL
LIN {X 0,Y 383.507,Z 290.336,A -85,B 0,C 180,E1 -11880.002,E2 -11880.002} C_VEL
LIN {X 0,Y 383.23,Z 290.375,A -85,B 0,C 180,E1 -11883.155,E2 -11883.155} C_VEL
LIN {X 0,Y 383.251,Z 290.37,A -85,B 0,C 180,E1 -11886.318,E2 -11886.318} C_VEL
LIN {X 0,Y 383.133,Z 290.384,A -85,B 0,C 180,E1 -11889.504,E2 -11889.504} C_VEL
LIN {X 0,Y 383.117,Z 290.383,A -85,B 0,C 180,E1 -11893.538,E2 -11893.538} C_VEL
LIN {X 0,Y 383.086,Z 290.387,A -85,B 0,C 180,E1 -11897.071,E2 -11897.071} C_VEL
LIN {X 0,Y 383.022,Z 290.397,A -85,B 0,C 180,E1 -11900.648,E2 -11900.648} C_VEL
LIN {X 0,Y 383.001,Z 290.398,A -85,B 0,C 180,E1 -11903.811,E2 -11903.811} C_VEL
LIN {X 0,Y 382.977,Z 290.403,A -85,B 0,C 180,E1 -11907.309,E2 -11907.309} C_VEL
LIN {X 0,Y 382.975,Z 290.4,A -85,B 0,C 180,E1 -11910.921,E2 -11910.921} C_VEL
LIN {X 0,Y 383.006,Z 290.398,A -85,B 0,C 180,E1 -11914.67,E2 -11914.67} C_VEL
LIN {X 0,Y 382.987,Z 290.403,A -85,B 0,C 180,E1 -11917.904,E2 -11917.904} C_VEL
LIN {X 0,Y 382.956,Z 290.404,A -85,B 0,C 180,E1 -11921.352,E2 -11921.352} C_VEL
LIN {X 0,Y 382.985,Z 290.405,A -85,B 0,C 180,E1 -11924.304,E2 -11924.304} C_VEL
LIN {X 0,Y 382.98,Z 290.404,A -85,B 0,C 180,E1 -11927.238,E2 -11927.238} C_VEL
LIN {X 0,Y 382.983,Z 290.406,A -85,B 0,C 180,E1 -11930.421,E2 -11930.421} C_VEL
LIN {X 0,Y 383.047,Z 290.59,A -85,B 0,C 180,E1 -11934.099,E2 -11934.099} C_VEL
LIN {X 0,Y 386.295,Z 302.377,A -85,B 0,C 180,E1 -11936.922,E2 -11936.922} C_VEL
LIN {X 0,Y 389.355,Z 314.537,A -85,B 0,C 180,E1 -11939.643,E2 -11939.643} C_VEL
LIN {X 0,Y 389.714,Z 316.284,A -85,B 0,C 180,E1 -11940.012,E2 -11940.012} C_VEL
LIN {X 0,Y 393.684,Z 325.789,A -85,B 0,C 180,E1 -11940.578,E2 -11940.578} C_VEL
LIN {X 0,Y 398.708,Z 351.587,A -85,B 0,C 180,E1 -11941.568,E2 -11941.568} C_VEL
LIN {X 0,Y 399.515,Z 356.612,A -85,B 0,C 180,E1 -11941.741,E2 -11941.741} C_VEL
LIN {X 0,Y 396.283,Z 483.477,A -85,B 0,C 180,E1 -11944.177,E2 -11944.177} C_VEL
LIN {X 0,Y 395.36,Z 499.18,A -85,B 0,C 180,E1 -11944.677,E2 -11944.677} C_VEL
LIN {X 0,Y 394.23,Z 513.216,A -85,B 0,C 180,E1 -11945.311,E2 -11945.311} C_VEL
LIN {X 0,Y 392.907,Z 526.948,A -85,B 0,C 180,E1 -11946.129,E2 -11946.129} C_VEL
LIN {X 0,Y 391.449,Z 540.578,A -85,B 0,C 180,E1 -11947.155,E2 -11947.155} C_VEL
LIN {X 0,Y 389.697,Z 554.442,A -85,B 0,C 180,E1 -11948.442,E2 -11948.442} C_VEL
LIN {X 0,Y 388.041,Z 567.004,A -85,B 0,C 180,E1 -11949.873,E2 -11949.873} C_VEL
LIN {X 0,Y 386.582,Z 578.46,A -85,B 0,C 180,E1 -11951.45,E2 -11951.45} C_VEL
LIN {X 0,Y 385.206,Z 588.112,A -85,B 0,C 180,E1 -11953.028,E2 -11953.028} C_VEL
LIN {X 0,Y 384.012,Z 597.613,A -85,B 0,C 180,E1 -11954.883,E2 -11954.883} C_VEL
LIN {X 0,Y 383.077,Z 605.944,A -85,B 0,C 180,E1 -11956.851,E2 -11956.851} C_VEL
LIN {X 0,Y 382.392,Z 612.942,A -85,B 0,C 180,E1 -11958.874,E2 -11958.874} C_VEL
LIN {X 0,Y 381.889,Z 618.818,A -85,B 0,C 180,E1 -11961.001,E2 -11961.001} C_VEL
LIN {X 0,Y 381.697,Z 622.325,A -85,B 0,C 180,E1 -11962.595,E2 -11962.595} C_VEL
LIN {X 0,Y 381.553,Z 625.849,A -85,B 0,C 180,E1 -11964.716,E2 -11964.716} C_VEL
LIN {X 0,Y 381.524,Z 628.157,A -85,B 0,C 180,E1 -11966.833,E2 -11966.833} C_VEL
LIN {X 0,Y 381.617,Z 629.298,A -85,B 0,C 180,E1 -11968.945,E2 -11968.945} C_VEL
LIN {X 0,Y 381.617,Z 629.28,A -85,B 0,C 180,E1 -11971.056,E2 -11971.056} C_VEL
LIN {X 0,Y 381.525,Z 628.042,A -85,B 0,C 180,E1 -11973.168,E2 -11973.168} C_VEL
LIN {X 0,Y 381.572,Z 625.627,A -85,B 0,C 180,E1 -11975.284,E2 -11975.284} C_VEL
LIN {X 0,Y 381.722,Z 621.985,A -85,B 0,C 180,E1 -11977.405,E2 -11977.405} C_VEL
LIN {X 0,Y 381.976,Z 617.021,A -85,B 0,C 180,E1 -11979.532,E2 -11979.532} C_VEL
LIN {X 0,Y 382.559,Z 610.608,A -85,B 0,C 180,E1 -11981.659,E2 -11981.659} C_VEL
LIN {X 0,Y 383.274,Z 602.557,A -85,B 0,C 180,E1 -11983.791,E2 -11983.791} C_VEL
LIN {X 0,Y 384.264,Z 593.971,A -85,B 0,C 180,E1 -11985.651,E2 -11985.651} C_VEL
LIN {X 0,Y 385.312,Z 585.265,A -85,B 0,C 180,E1 -11987.241,E2 -11987.241} C_VEL
LIN {X 0,Y 386.662,Z 574.981,A -85,B 0,C 180,E1 -11988.818,E2 -11988.818} C_VEL
LIN {X 0,Y 388.118,Z 562.664,A -85,B 0,C 180,E1 -11990.4,E2 -11990.4} C_VEL
LIN {X 0,Y 389.675,Z 550.336,A -85,B 0,C 180,E1 -11991.699,E2 -11991.699} C_VEL
LIN {X 0,Y 391.19,Z 536.914,A -85,B 0,C 180,E1 -11992.862,E2 -11992.862} C_VEL
LIN {X 0,Y 392.51,Z 523.535,A -85,B 0,C 180,E1 -11993.797,E2 -11993.797} C_VEL
LIN {X 0,Y 393.676,Z 509.058,A -85,B 0,C 180,E1 -11994.594,E2 -11994.594} C_VEL
LIN {X 0,Y 394.705,Z 494.197,A -85,B 0,C 180,E1 -11995.193,E2 -11995.193} C_VEL
LIN {X 0,Y 395.392,Z 479.073,A -85,B 0,C 180,E1 -11995.604,E2 -11995.604} C_VEL
LIN {X 0,Y 398.139,Z 355.521,A -85,B 0,C 180,E1 -11997.939,E2 -11997.939} C_VEL
LIN {X 0,Y 391.876,Z 322.88,A -85,B 0,C 180,E1 -11999.081,E2 -11999.081} C_VEL
LIN {X 0,Y 389.647,Z 317.088,A -85,B 0,C 180,E1 -11999.404,E2 -11999.404} C_VEL
LIN {X 0,Y 386.187,Z 302.592,A -85,B 0,C 180,E1 -12002.447,E2 -12002.447} C_VEL
LIN {X 0,Y 383.03,Z 290.403,A -85,B 0,C 180,E1 -12005.147,E2 -12005.147} C_VEL
LIN {X 0,Y 382.982,Z 290.406,A -85,B 0,C 180,E1 -12008.603,E2 -12008.603} C_VEL
LIN {X 0,Y 382.962,Z 290.405,A -85,B 0,C 180,E1 -12011.35,E2 -12011.35} C_VEL
LIN {X 0,Y 382.989,Z 290.403,A -85,B 0,C 180,E1 -12014.301,E2 -12014.301} C_VEL
LIN {X 0,Y 382.983,Z 290.401,A -85,B 0,C 180,E1 -12017.235,E2 -12017.235} C_VEL
LIN {X 0,Y 382.985,Z 290.398,A -85,B 0,C 180,E1 -12020.418,E2 -12020.418} C_VEL
LIN {X 0,Y 383.012,Z 290.399,A -85,B 0,C 180,E1 -12024.042,E2 -12024.042} C_VEL
LIN {X 0,Y 382.985,Z 290.402,A -85,B 0,C 180,E1 -12027.577,E2 -12027.577} C_VEL
LIN {X 0,Y 382.975,Z 290.405,A -85,B 0,C 180,E1 -12030.297,E2 -12030.297} C_VEL
LIN {X 0,Y 383.001,Z 290.406,A -85,B 0,C 180,E1 -12034.044,E2 -12034.044} C_VEL
LIN {X 0,Y 382.984,Z 290.403,A -85,B 0,C 180,E1 -12037.332,E2 -12037.332} C_VEL
LIN {X 0,Y 383.055,Z 290.391,A -85,B 0,C 180,E1 -12040.715,E2 -12040.715} C_VEL
LIN {X 0,Y 383.075,Z 290.39,A -85,B 0,C 180,E1 -12044.025,E2 -12044.025} C_VEL
LIN {X 0,Y 383.13,Z 290.36,A -85,B 0,C 180,E1 -12047.282,E2 -12047.282} C_VEL
LIN {X 0,Y 383.131,Z 290.38,A -85,B 0,C 180,E1 -12050.496,E2 -12050.496} C_VEL
LIN {X 0,Y 383.227,Z 290.37,A -85,B 0,C 180,E1 -12053.681,E2 -12053.681} C_VEL
LIN {X 0,Y 383.358,Z 290.338,A -85,B 0,C 180,E1 -12057.897,E2 -12057.897} C_VEL
LIN {X 0,Y 383.368,Z 290.353,A -85,B 0,C 180,E1 -12062.099,E2 -12062.099} C_VEL
LIN {X 0,Y 383.19,Z 290.347,A -85,B 0,C 180,E1 -12066.409,E2 -12066.409} C_VEL
LIN {X 0,Y 383.112,Z 290.381,A -85,B 0,C 180,E1 -12069.501,E2 -12069.501} C_VEL
LIN {X 0,Y 383.127,Z 290.384,A -85,B 0,C 180,E1 -12072.714,E2 -12072.714} C_VEL
LIN {X 0,Y 383.065,Z 290.368,A -85,B 0,C 180,E1 -12075.972,E2 -12075.972} C_VEL
LIN {X 0,Y 383.047,Z 290.383,A -85,B 0,C 180,E1 -12079.282,E2 -12079.282} C_VEL
LIN {X 0,Y 382.979,Z 290.402,A -85,B 0,C 180,E1 -12082.664,E2 -12082.664} C_VEL
LIN {X 0,Y 382.97,Z 290.383,A -85,B 0,C 180,E1 -12086.129,E2 -12086.129} C_VEL
LIN {X 0,Y 382.963,Z 290.402,A -85,B 0,C 180,E1 -12089.7,E2 -12089.7} C_VEL
LIN {X 0,Y 382.986,Z 290.4,A -85,B 0,C 180,E1 -12093.4,E2 -12093.4} C_VEL
LIN {X 0,Y 383.009,Z 290.378,A -85,B 0,C 180,E1 -12096.161,E2 -12096.161} C_VEL
LIN {X 0,Y 382.971,Z 290.404,A -85,B 0,C 180,E1 -12099.579,E2 -12099.579} C_VEL
LIN {X 0,Y 382.992,Z 290.403,A -85,B 0,C 180,E1 -12102.777,E2 -12102.777} C_VEL
LIN {X 0,Y 382.98,Z 290.388,A -85,B 0,C 180,E1 -12105.787,E2 -12105.787} C_VEL
LIN {X 0,Y 382.97,Z 290.407,A -85,B 0,C 180,E1 -12108.795,E2 -12108.795} C_VEL
LIN {X 0,Y 382.982,Z 290.394,A -85,B 0,C 180,E1 -12112.095,E2 -12112.095} C_VEL
LIN {X 0,Y 383.002,Z 290.403,A -85,B 0,C 180,E1 -12115.331,E2 -12115.331} C_VEL
LIN {X 0,Y 382.966,Z 290.394,A -85,B 0,C 180,E1 -12119.08,E2 -12119.08} C_VEL
LIN {X 0,Y 383.04,Z 290.399,A -85,B 0,C 180,E1 -12122.697,E2 -12122.697} C_VEL
LIN {X 0,Y 383.032,Z 290.39,A -85,B 0,C 180,E1 -12125.039,E2 -12125.039} C_VEL
LIN {X 0,Y 382.975,Z 290.406,A -85,B 0,C 180,E1 -12128.468,E2 -12128.468} C_VEL
LIN {X 0,Y 383.045,Z 290.396,A -85,B 0,C 180,E1 -12131.826,E2 -12131.826} C_VEL
LIN {X 0,Y 383.094,Z 290.391,A -85,B 0,C 180,E1 -12135.118,E2 -12135.118} C_VEL
LIN {X 0,Y 383.091,Z 290.392,A -85,B 0,C 180,E1 -12138.358,E2 -12138.358} C_VEL
LIN {X 0,Y 383.246,Z 290.368,A -85,B 0,C 180,E1 -12141.975,E2 -12141.975} C_VEL
LIN {X 0,Y 383.178,Z 290.381,A -85,B 0,C 180,E1 -12144.738,E2 -12144.738} C_VEL
LIN {X 0,Y 383.324,Z 290.355,A -85,B 0,C 180,E1 -12148.555,E2 -12148.555} C_VEL
LIN {X 0,Y 385.24,Z 298.018,A -85,B 0,C 180,E1 -12150.352,E2 -12150.352} C_VEL
LIN {X 0,Y 394.375,Z 319.211,A -85,B 0,C 180,E1 -12151.514,E2 -12151.514} C_VEL
LIN {X 0,Y 398.457,Z 329.061,A -85,B 0,C 180,E1 -12152.021,E2 -12152.021} C_VEL
LIN {X 0,Y 396.866,Z 404.931,A -85,B 0,C 180,E1 -12153.458,E2 -12153.458} C_VEL
LIN {X 0,Y 395.517,Z 463.005,A -85,B 0,C 180,E1 -12154.575,E2 -12154.575} C_VEL
LIN {X 0,Y 394.766,Z 478.672,A -85,B 0,C 180,E1 -12155.078,E2 -12155.078} C_VEL
LIN {X 0,Y 393.75,Z 493.52,A -85,B 0,C 180,E1 -12155.762,E2 -12155.762} C_VEL
LIN {X 0,Y 392.682,Z 506.564,A -85,B 0,C 180,E1 -12156.553,E2 -12156.553} C_VEL
LIN {X 0,Y 391.565,Z 511.925,A -85,B 0,C 180,E1 -12156.895,E2 -12156.895} C_VEL
LIN {X 0,Y 388.035,Z 520.539,A -85,B 0,C 180,E1 -12157.42,E2 -12157.42} C_VEL
LIN {X 0,Y 384.438,Z 528.816,A -85,B 0,C 180,E1 -12158.012,E2 -12158.012} C_VEL
LIN {X 0,Y 383.188,Z 533.65,A -85,B 0,C 180,E1 -12158.465,E2 -12158.465} C_VEL
LIN {X 0,Y 381.597,Z 546.385,A -85,B 0,C 180,E1 -12159.942,E2 -12159.942} C_VEL
LIN {X 0,Y 380.125,Z 557.643,A -85,B 0,C 180,E1 -12161.521,E2 -12161.521} C_VEL
LIN {X 0,Y 378.81,Z 567.292,A -85,B 0,C 180,E1 -12163.136,E2 -12163.136} C_VEL
LIN {X 0,Y 377.642,Z 575.833,A -85,B 0,C 180,E1 -12164.827,E2 -12164.827} C_VEL
LIN {X 0,Y 376.592,Z 584.18,A -85,B 0,C 180,E1 -12166.813,E2 -12166.813} C_VEL
LIN {X 0,Y 375.907,Z 590.206,A -85,B 0,C 180,E1 -12168.531,E2 -12168.531} C_VEL
LIN {X 0,Y 375.215,Z 596.708,A -85,B 0,C 180,E1 -12170.846,E2 -12170.846} C_VEL
LIN {X 0,Y 374.817,Z 601.643,A -85,B 0,C 180,E1 -12173.188,E2 -12173.188} C_VEL
LIN {X 0,Y 374.429,Z 605.148,A -85,B 0,C 180,E1 -12175.575,E2 -12175.575} C_VEL
LIN {X 0,Y 374.275,Z 607.212,A -85,B 0,C 180,E1 -12177.997,E2 -12177.997} C_VEL
LIN {X 0,Y 374.213,Z 607.818,A -85,B 0,C 180,E1 -12180.468,E2 -12180.468} C_VEL
LIN {X 0,Y 374.302,Z 607.283,A -85,B 0,C 180,E1 -12182.34,E2 -12182.34} C_VEL
LIN {X 0,Y 374.423,Z 605.752,A -85,B 0,C 180,E1 -12184.326,E2 -12184.326} C_VEL
LIN {X 0,Y 374.702,Z 603.366,A -85,B 0,C 180,E1 -12186.247,E2 -12186.247} C_VEL
LIN {X 0,Y 375.058,Z 599.903,A -85,B 0,C 180,E1 -12188.196,E2 -12188.196} C_VEL
LIN {X 0,Y 375.589,Z 594.883,A -85,B 0,C 180,E1 -12190.341,E2 -12190.341} C_VEL
LIN {X 0,Y 376.295,Z 589.243,A -85,B 0,C 180,E1 -12192.248,E2 -12192.248} C_VEL
LIN {X 0,Y 377.273,Z 581.738,A -85,B 0,C 180,E1 -12194.31,E2 -12194.31} C_VEL
LIN {X 0,Y 378.357,Z 574.184,A -85,B 0,C 180,E1 -12196.035,E2 -12196.035} C_VEL
LIN {X 0,Y 379.643,Z 565.11,A -85,B 0,C 180,E1 -12197.771,E2 -12197.771} C_VEL
LIN {X 0,Y 381.293,Z 554.145,A -85,B 0,C 180,E1 -12199.516,E2 -12199.516} C_VEL
LIN {X 0,Y 382.885,Z 542.72,A -85,B 0,C 180,E1 -12201.027,E2 -12201.027} C_VEL
LIN {X 0,Y 384.628,Z 529.939,A -85,B 0,C 180,E1 -12202.423,E2 -12202.423} C_VEL
LIN {X 0,Y 386.219,Z 516.452,A -85,B 0,C 180,E1 -12203.628,E2 -12203.628} C_VEL
LIN {X 0,Y 387.723,Z 502.069,A -85,B 0,C 180,E1 -12204.653,E2 -12204.653} C_VEL
LIN {X 0,Y 389.041,Z 486.452,A -85,B 0,C 180,E1 -12205.506,E2 -12205.506} C_VEL
LIN {X 0,Y 390,Z 471.293,A -85,B 0,C 180,E1 -12206.103,E2 -12206.103} C_VEL
LIN {X 0,Y 390.621,Z 454.849,A -85,B 0,C 180,E1 -12206.521,E2 -12206.521} C_VEL
LIN {X 0,Y 393.821,Z 332.38,A -85,B 0,C 180,E1 -12208.903,E2 -12208.903} C_VEL
LIN {X 0,Y 386.69,Z 316.293,A -85,B 0,C 180,E1 -12209.903,E2 -12209.903} C_VEL
LIN {X 0,Y 379.006,Z 301.048,A -85,B 0,C 180,E1 -12211,E2 -12211} C_VEL
LIN {X 0,Y 378.116,Z 299.05,A -85,B 0,C 180,E1 -12211.157,E2 -12211.157} C_VEL
LIN {X 0,Y 376.013,Z 291.27,A -85,B 0,C 180,E1 -12213.275,E2 -12213.275} C_VEL
LIN {X 0,Y 375.981,Z 291.28,A -85,B 0,C 180,E1 -12216.89,E2 -12216.89} C_VEL
LIN {X 0,Y 375.983,Z 291.274,A -85,B 0,C 180,E1 -12220.341,E2 -12220.341} C_VEL
LIN {X 0,Y 376.015,Z 291.274,A -85,B 0,C 180,E1 -12223.72,E2 -12223.72} C_VEL
LIN {X 0,Y 376.09,Z 291.262,A -85,B 0,C 180,E1 -12227.044,E2 -12227.044} C_VEL
LIN {X 0,Y 376.106,Z 291.26,A -85,B 0,C 180,E1 -12230.32,E2 -12230.32} C_VEL
LIN {X 0,Y 376.228,Z 291.242,A -85,B 0,C 180,E1 -12233.567,E2 -12233.567} C_VEL
LIN {X 0,Y 376.34,Z 291.231,A -85,B 0,C 180,E1 -12237.861,E2 -12237.861} C_VEL
LIN {X 0,Y 376.477,Z 291.212,A -85,B 0,C 180,E1 -12240.002,E2 -12240.002} C_VEL
LIN {X 0,Y 376.168,Z 291.254,A -85,B 0,C 180,E1 -12243.215,E2 -12243.215} C_VEL
LIN {X 0,Y 376.21,Z 291.248,A -85,B 0,C 180,E1 -12246.437,E2 -12246.437} C_VEL
LIN {X 0,Y 376.104,Z 291.26,A -85,B 0,C 180,E1 -12249.683,E2 -12249.683} C_VEL
LIN {X 0,Y 376.082,Z 291.259,A -85,B 0,C 180,E1 -12253.659,E2 -12253.659} C_VEL
LIN {X 0,Y 376.025,Z 291.267,A -85,B 0,C 180,E1 -12257.402,E2 -12257.402} C_VEL
LIN {X 0,Y 375.972,Z 291.277,A -85,B 0,C 180,E1 -12260.834,E2 -12260.834} C_VEL
LIN {X 0,Y 375.951,Z 291.279,A -85,B 0,C 180,E1 -12264.286,E2 -12264.286} C_VEL
LIN {X 0,Y 375.921,Z 291.283,A -85,B 0,C 180,E1 -12267.866,E2 -12267.866} C_VEL
LIN {X 0,Y 375.932,Z 291.279,A -85,B 0,C 180,E1 -12270.691,E2 -12270.691} C_VEL
LIN {X 0,Y 375.952,Z 291.276,A -85,B 0,C 180,E1 -12274.114,E2 -12274.114} C_VEL
LIN {X 0,Y 375.943,Z 291.276,A -85,B 0,C 180,E1 -12276.744,E2 -12276.744} C_VEL
LIN {X 0,Y 375.934,Z 291.28,A -85,B 0,C 180,E1 -12279.963,E2 -12279.963} C_VEL
LIN {X 0,Y 375.921,Z 291.282,A -85,B 0,C 180,E1 -12283.769,E2 -12283.769} C_VEL
LIN {X 0,Y 375.93,Z 291.283,A -85,B 0,C 180,E1 -12286.813,E2 -12286.813} C_VEL
LIN {X 0,Y 375.932,Z 291.284,A -85,B 0,C 180,E1 -12290.535,E2 -12290.535} C_VEL
LIN {X 0,Y 375.977,Z 291.344,A -85,B 0,C 180,E1 -12293.45,E2 -12293.45} C_VEL
LIN {X 0,Y 379.124,Z 302.465,A -85,B 0,C 180,E1 -12296.213,E2 -12296.213} C_VEL
LIN {X 0,Y 382.476,Z 315.861,A -85,B 0,C 180,E1 -12299.297,E2 -12299.297} C_VEL
LIN {X 0,Y 387.881,Z 328.461,A -85,B 0,C 180,E1 -12300.118,E2 -12300.118} C_VEL
LIN {X 0,Y 392.445,Z 352.066,A -85,B 0,C 180,E1 -12301.045,E2 -12301.045} C_VEL
LIN {X 0,Y 393.329,Z 358.255,A -85,B 0,C 180,E1 -12301.257,E2 -12301.257} C_VEL
LIN {X 0,Y 389.979,Z 482.943,A -85,B 0,C 180,E1 -12303.692,E2 -12303.692} C_VEL
LIN {X 0,Y 388.997,Z 498.755,A -85,B 0,C 180,E1 -12304.197,E2 -12304.197} C_VEL
LIN {X 0,Y 387.836,Z 513.064,A -85,B 0,C 180,E1 -12304.854,E2 -12304.854} C_VEL
LIN {X 0,Y 386.414,Z 527.196,A -85,B 0,C 180,E1 -12305.71,E2 -12305.71} C_VEL
LIN {X 0,Y 384.9,Z 540.645,A -85,B 0,C 180,E1 -12306.744,E2 -12306.744} C_VEL
LIN {X 0,Y 383.082,Z 554.459,A -85,B 0,C 180,E1 -12308.051,E2 -12308.051} C_VEL
LIN {X 0,Y 381.349,Z 566.977,A -85,B 0,C 180,E1 -12309.504,E2 -12309.504} C_VEL
LIN {X 0,Y 379.789,Z 578.386,A -85,B 0,C 180,E1 -12311.106,E2 -12311.106} C_VEL
LIN {X 0,Y 378.358,Z 588.004,A -85,B 0,C 180,E1 -12312.711,E2 -12312.711} C_VEL
LIN {X 0,Y 377.104,Z 597.488,A -85,B 0,C 180,E1 -12314.6,E2 -12314.6} C_VEL
LIN {X 0,Y 376.095,Z 605.47,A -85,B 0,C 180,E1 -12316.513,E2 -12316.513} C_VEL
LIN {X 0,Y 375.379,Z 612.791,A -85,B 0,C 180,E1 -12318.663,E2 -12318.663} C_VEL
LIN {X 0,Y 374.827,Z 618.656,A -85,B 0,C 180,E1 -12320.83,E2 -12320.83} C_VEL
LIN {X 0,Y 374.631,Z 622.159,A -85,B 0,C 180,E1 -12322.455,E2 -12322.455} C_VEL
LIN {X 0,Y 374.466,Z 625.67,A -85,B 0,C 180,E1 -12324.616,E2 -12324.616} C_VEL
LIN {X 0,Y 374.438,Z 627.967,A -85,B 0,C 180,E1 -12326.773,E2 -12326.773} C_VEL
LIN {X 0,Y 374.516,Z 629.097,A -85,B 0,C 180,E1 -12328.925,E2 -12328.925} C_VEL
LIN {X 0,Y 374.517,Z 629.071,A -85,B 0,C 180,E1 -12331.076,E2 -12331.076} C_VEL
LIN {X 0,Y 374.44,Z 627.824,A -85,B 0,C 180,E1 -12333.228,E2 -12333.228} C_VEL
LIN {X 0,Y 374.49,Z 625.396,A -85,B 0,C 180,E1 -12335.385,E2 -12335.385} C_VEL
LIN {X 0,Y 374.647,Z 621.738,A -85,B 0,C 180,E1 -12337.546,E2 -12337.546} C_VEL
LIN {X 0,Y 374.912,Z 616.754,A -85,B 0,C 180,E1 -12339.713,E2 -12339.713} C_VEL
LIN {X 0,Y 375.545,Z 610.318,A -85,B 0,C 180,E1 -12341.88,E2 -12341.88} C_VEL
LIN {X 0,Y 376.305,Z 602.239,A -85,B 0,C 180,E1 -12344.052,E2 -12344.052} C_VEL
LIN {X 0,Y 377.329,Z 593.624,A -85,B 0,C 180,E1 -12345.946,E2 -12345.946} C_VEL
LIN {X 0,Y 378.494,Z 584.893,A -85,B 0,C 180,E1 -12347.562,E2 -12347.562} C_VEL
LIN {X 0,Y 379.854,Z 574.447,A -85,B 0,C 180,E1 -12349.189,E2 -12349.189} C_VEL
LIN {X 0,Y 381.373,Z 562.22,A -85,B 0,C 180,E1 -12350.778,E2 -12350.778} C_VEL
LIN {X 0,Y 383.032,Z 549.851,A -85,B 0,C 180,E1 -12352.095,E2 -12352.095} C_VEL
LIN {X 0,Y 384.574,Z 536.362,A -85,B 0,C 180,E1 -12353.278,E2 -12353.278} C_VEL
LIN {X 0,Y 386.047,Z 522.151,A -85,B 0,C 180,E1 -12354.274,E2 -12354.274} C_VEL
LIN {X 0,Y 387.295,Z 506.991,A -85,B 0,C 180,E1 -12355.098,E2 -12355.098} C_VEL
LIN {X 0,Y 388.382,Z 491.371,A -85,B 0,C 180,E1 -12355.704,E2 -12355.704} C_VEL
LIN {X 0,Y 389.024,Z 476.122,A -85,B 0,C 180,E1 -12356.09,E2 -12356.09} C_VEL
LIN {X 0,Y 391.796,Z 356.899,A -85,B 0,C 180,E1 -12358.371,E2 -12358.371} C_VEL
LIN {X 0,Y 385.94,Z 325.747,A -85,B 0,C 180,E1 -12359.478,E2 -12359.478} C_VEL
LIN {X 0,Y 382.414,Z 316.969,A -85,B 0,C 180,E1 -12359.962,E2 -12359.962} C_VEL
LIN {X 0,Y 379.252,Z 303.891,A -85,B 0,C 180,E1 -12362.775,E2 -12362.775} C_VEL
LIN {X 0,Y 375.995,Z 291.276,A -85,B 0,C 180,E1 -12365.658,E2 -12365.658} C_VEL
LIN {X 0,Y 375.935,Z 291.286,A -85,B 0,C 180,E1 -12369.465,E2 -12369.465} C_VEL
LIN {X 0,Y 375.933,Z 291.276,A -85,B 0,C 180,E1 -12373.188,E2 -12373.188} C_VEL
LIN {X 0,Y 375.933,Z 291.278,A -85,B 0,C 180,E1 -12376.81,E2 -12376.81} C_VEL
LIN {X 0,Y 375.934,Z 291.276,A -85,B 0,C 180,E1 -12380.532,E2 -12380.532} C_VEL
LIN {X 0,Y 375.957,Z 291.284,A -85,B 0,C 180,E1 -12383.496,E2 -12383.496} C_VEL
LIN {X 0,Y 375.957,Z 291.269,A -85,B 0,C 180,E1 -12385.887,E2 -12385.887} C_VEL
LIN {X 0,Y 375.961,Z 291.277,A -85,B 0,C 180,E1 -12389.686,E2 -12389.686} C_VEL
LIN {X 0,Y 375.916,Z 291.282,A -85,B 0,C 180,E1 -12392.134,E2 -12392.134} C_VEL
LIN {X 0,Y 375.956,Z 291.282,A -85,B 0,C 180,E1 -12395.715,E2 -12395.715} C_VEL
LIN {X 0,Y 375.978,Z 291.279,A -85,B 0,C 180,E1 -12399.195,E2 -12399.195} C_VEL
LIN {X 0,Y 376.03,Z 291.271,A -85,B 0,C 180,E1 -12402.599,E2 -12402.599} C_VEL
LIN {X 0,Y 376.087,Z 291.24,A -85,B 0,C 180,E1 -12406.341,E2 -12406.341} C_VEL
LIN {X 0,Y 376.102,Z 291.256,A -85,B 0,C 180,E1 -12410.317,E2 -12410.317} C_VEL
LIN {X 0,Y 376.187,Z 291.248,A -85,B 0,C 180,E1 -12413.562,E2 -12413.562} C_VEL
LIN {X 0,Y 376.322,Z 291.213,A -85,B 0,C 180,E1 -12417.858,E2 -12417.858} C_VEL
LIN {X 0,Y 376.333,Z 291.229,A -85,B 0,C 180,E1 -12422.139,E2 -12422.139} C_VEL
LIN {X 0,Y 376.16,Z 291.222,A -85,B 0,C 180,E1 -12426.435,E2 -12426.435} C_VEL
LIN {X 0,Y 376.096,Z 291.247,A -85,B 0,C 180,E1 -12428.596,E2 -12428.596} C_VEL
LIN {X 0,Y 376.037,Z 291.268,A -85,B 0,C 180,E1 -12431.862,E2 -12431.862} C_VEL
LIN {X 0,Y 376.043,Z 291.251,A -85,B 0,C 180,E1 -12435.166,E2 -12435.166} C_VEL
LIN {X 0,Y 375.992,Z 291.255,A -85,B 0,C 180,E1 -12438.525,E2 -12438.525} C_VEL
LIN {X 0,Y 375.948,Z 291.278,A -85,B 0,C 180,E1 -12441.953,E2 -12441.953} C_VEL
LIN {X 0,Y 375.924,Z 291.264,A -85,B 0,C 180,E1 -12445.465,E2 -12445.465} C_VEL
LIN {X 0,Y 375.901,Z 291.271,A -85,B 0,C 180,E1 -12449.082,E2 -12449.082} C_VEL
LIN {X 0,Y 375.944,Z 291.281,A -85,B 0,C 180,E1 -12451.561,E2 -12451.561} C_VEL
LIN {X 0,Y 375.936,Z 291.262,A -85,B 0,C 180,E1 -12455.415,E2 -12455.415} C_VEL
LIN {X 0,Y 375.921,Z 291.269,A -85,B 0,C 180,E1 -12458.261,E2 -12458.261} C_VEL
LIN {X 0,Y 375.903,Z 291.285,A -85,B 0,C 180,E1 -12461.596,E2 -12461.596} C_VEL
LIN {X 0,Y 375.907,Z 291.269,A -85,B 0,C 180,E1 -12464.729,E2 -12464.729} C_VEL
LIN {X 0,Y 375.917,Z 291.282,A -85,B 0,C 180,E1 -12468.398,E2 -12468.398} C_VEL
LIN {X 0,Y 375.956,Z 291.27,A -85,B 0,C 180,E1 -12471.729,E2 -12471.729} C_VEL
LIN {X 0,Y 375.964,Z 291.28,A -85,B 0,C 180,E1 -12475.332,E2 -12475.332} C_VEL
LIN {X 0,Y 375.941,Z 291.276,A -85,B 0,C 180,E1 -12478.437,E2 -12478.437} C_VEL
LIN {X 0,Y 375.965,Z 291.276,A -85,B 0,C 180,E1 -12482.139,E2 -12482.139} C_VEL
LIN {X 0,Y 375.988,Z 291.268,A -85,B 0,C 180,E1 -12484.538,E2 -12484.538} C_VEL
LIN {X 0,Y 375.939,Z 291.281,A -85,B 0,C 180,E1 -12488.044,E2 -12488.044} C_VEL
LIN {X 0,Y 375.992,Z 291.275,A -85,B 0,C 180,E1 -12491.472,E2 -12491.472} C_VEL
LIN {X 0,Y 376.042,Z 291.27,A -85,B 0,C 180,E1 -12494.832,E2 -12494.832} C_VEL
LIN {X 0,Y 376.042,Z 291.269,A -85,B 0,C 180,E1 -12498.136,E2 -12498.136} C_VEL
LIN {X 0,Y 376.201,Z 291.246,A -85,B 0,C 180,E1 -12501.918,E2 -12501.918} C_VEL
LIN {X 0,Y 376.151,Z 291.255,A -85,B 0,C 180,E1 -12504.639,E2 -12504.639} C_VEL
LIN {X 0,Y 376.32,Z 291.338,A -85,B 0,C 180,E1 -12508.127,E2 -12508.127} C_VEL
LIN {X 0,Y 378.092,Z 298.212,A -85,B 0,C 180,E1 -12509.775,E2 -12509.775} C_VEL
LIN {X 0,Y 387.965,Z 320.814,A -85,B 0,C 180,E1 -12511.057,E2 -12511.057} C_VEL
LIN {X 0,Y 392.192,Z 330.803,A -85,B 0,C 180,E1 -12511.593,E2 -12511.593} C_VEL
LIN {X 0,Y 389.051,Z 462.926,A -85,B 0,C 180,E1 -12514.143,E2 -12514.143} C_VEL
LIN {X 0,Y 388.291,Z 478.511,A -85,B 0,C 180,E1 -12514.647,E2 -12514.647} C_VEL
LIN {X 0,Y 387.246,Z 493.357,A -85,B 0,C 180,E1 -12515.336,E2 -12515.336} C_VEL
LIN {X 0,Y 385.948,Z 508.404,A -85,B 0,C 180,E1 -12516.272,E2 -12516.272} C_VEL
LIN {X 0,Y 384.532,Z 522.08,A -85,B 0,C 180,E1 -12517.35,E2 -12517.35} C_VEL
LIN {X 0,Y 383.188,Z 533.65,A -85,B 0,C 180,E1 -12518.465,E2 -12518.465} C_VEL
LIN {X 0,Y 381.944,Z 538.461,A -85,B 0,C 180,E1 -12518.945,E2 -12518.945} C_VEL
LIN {X 0,Y 378.261,Z 546.098,A -85,B 0,C 180,E1 -12519.72,E2 -12519.72} C_VEL
LIN {X 0,Y 374.593,Z 553.426,A -85,B 0,C 180,E1 -12520.568,E2 -12520.568} C_VEL
LIN {X 0,Y 373.351,Z 557.638,A -85,B 0,C 180,E1 -12521.172,E2 -12521.172} C_VEL
LIN {X 0,Y 371.959,Z 567.391,A -85,B 0,C 180,E1 -12522.826,E2 -12522.826} C_VEL
LIN {X 0,Y 370.616,Z 576.843,A -85,B 0,C 180,E1 -12524.746,E2 -12524.746} C_VEL
LIN {X 0,Y 369.481,Z 585.388,A -85,B 0,C 180,E1 -12526.862,E2 -12526.862} C_VEL
LIN {X 0,Y 368.692,Z 592.092,A -85,B 0,C 180,E1 -12528.907,E2 -12528.907} C_VEL
LIN {X 0,Y 368.051,Z 598.208,A -85,B 0,C 180,E1 -12531.272,E2 -12531.272} C_VEL
LIN {X 0,Y 367.626,Z 602.803,A -85,B 0,C 180,E1 -12533.669,E2 -12533.669} C_VEL
LIN {X 0,Y 367.285,Z 605.965,A -85,B 0,C 180,E1 -12536.109,E2 -12536.109} C_VEL
LIN {X 0,Y 367.157,Z 607.688,A -85,B 0,C 180,E1 -12538.589,E2 -12538.589} C_VEL
LIN {X 0,Y 367.137,Z 607.94,A -85,B 0,C 180,E1 -12541.12,E2 -12541.12} C_VEL
LIN {X 0,Y 367.222,Z 607.384,A -85,B 0,C 180,E1 -12542.644,E2 -12542.644} C_VEL
LIN {X 0,Y 367.416,Z 605.37,A -85,B 0,C 180,E1 -12545.017,E2 -12545.017} C_VEL
LIN {X 0,Y 367.682,Z 603.224,A -85,B 0,C 180,E1 -12546.606,E2 -12546.606} C_VEL
LIN {X 0,Y 368.025,Z 599.925,A -85,B 0,C 180,E1 -12548.472,E2 -12548.472} C_VEL
LIN {X 0,Y 368.53,Z 595.454,A -85,B 0,C 180,E1 -12550.419,E2 -12550.419} C_VEL
LIN {X 0,Y 369.384,Z 589.215,A -85,B 0,C 180,E1 -12552.578,E2 -12552.578} C_VEL
LIN {X 0,Y 370.376,Z 582.007,A -85,B 0,C 180,E1 -12554.593,E2 -12554.593} C_VEL
LIN {X 0,Y 371.529,Z 574.474,A -85,B 0,C 180,E1 -12556.347,E2 -12556.347} C_VEL
LIN {X 0,Y 373.039,Z 564.423,A -85,B 0,C 180,E1 -12558.289,E2 -12558.289} C_VEL
LIN {X 0,Y 374.775,Z 553.417,A -85,B 0,C 180,E1 -12560.039,E2 -12560.039} C_VEL
LIN {X 0,Y 376.537,Z 541.435,A -85,B 0,C 180,E1 -12561.619,E2 -12561.619} C_VEL
LIN {X 0,Y 378.323,Z 528.57,A -85,B 0,C 180,E1 -12563.013,E2 -12563.013} C_VEL
LIN {X 0,Y 379.944,Z 515.424,A -85,B 0,C 180,E1 -12564.181,E2 -12564.181} C_VEL
LIN {X 0,Y 381.444,Z 501.496,A -85,B 0,C 180,E1 -12565.171,E2 -12565.171} C_VEL
LIN {X 0,Y 382.656,Z 487.48,A -85,B 0,C 180,E1 -12565.948,E2 -12565.948} C_VEL
LIN {X 0,Y 383.71,Z 471.794,A -85,B 0,C 180,E1 -12566.585,E2 -12566.585} C_VEL
LIN {X 0,Y 384.397,Z 455.974,A -85,B 0,C 180,E1 -12566.998,E2 -12566.998} C_VEL
LIN {X 0,Y 387.665,Z 334.213,A -85,B 0,C 180,E1 -12569.409,E2 -12569.409} C_VEL
LIN {X 0,Y 380.724,Z 318.709,A -85,B 0,C 180,E1 -12570.417,E2 -12570.417} C_VEL
LIN {X 0,Y 372.904,Z 303.108,A -85,B 0,C 180,E1 -12571.578,E2 -12571.578} C_VEL
LIN {X 0,Y 370.958,Z 299.36,A -85,B 0,C 180,E1 -12571.886,E2 -12571.886} C_VEL
LIN {X 0,Y 368.988,Z 292.148,A -85,B 0,C 180,E1 -12573.928,E2 -12573.928} C_VEL
LIN {X 0,Y 368.917,Z 292.154,A -85,B 0,C 180,E1 -12577.606,E2 -12577.606} C_VEL
LIN {X 0,Y 368.952,Z 292.147,A -85,B 0,C 180,E1 -12581.108,E2 -12581.108} C_VEL
LIN {X 0,Y 368.984,Z 292.15,A -85,B 0,C 180,E1 -12584.537,E2 -12584.537} C_VEL
LIN {X 0,Y 368.992,Z 292.147,A -85,B 0,C 180,E1 -12587.908,E2 -12587.908} C_VEL
LIN {X 0,Y 369.155,Z 292.125,A -85,B 0,C 180,E1 -12591.87,E2 -12591.87} C_VEL
LIN {X 0,Y 369.129,Z 292.127,A -85,B 0,C 180,E1 -12594.539,E2 -12594.539} C_VEL
LIN {X 0,Y 369.305,Z 292.107,A -85,B 0,C 180,E1 -12597.821,E2 -12597.821} C_VEL
LIN {X 0,Y 369.447,Z 292.088,A -85,B 0,C 180,E1 -12600.002,E2 -12600.002} C_VEL
LIN {X 0,Y 369.304,Z 292.102,A -85,B 0,C 180,E1 -12602.183,E2 -12602.183} C_VEL
LIN {X 0,Y 369.17,Z 292.126,A -85,B 0,C 180,E1 -12606.561,E2 -12606.561} C_VEL
LIN {X 0,Y 369.054,Z 292.138,A -85,B 0,C 180,E1 -12609.87,E2 -12609.87} C_VEL
LIN {X 0,Y 369.029,Z 292.137,A -85,B 0,C 180,E1 -12613.774,E2 -12613.774} C_VEL
LIN {X 0,Y 368.984,Z 292.144,A -85,B 0,C 180,E1 -12617.745,E2 -12617.745} C_VEL
LIN {X 0,Y 368.903,Z 292.158,A -85,B 0,C 180,E1 -12621.223,E2 -12621.223} C_VEL
LIN {X 0,Y 368.909,Z 292.153,A -85,B 0,C 180,E1 -12623.878,E2 -12623.878} C_VEL
LIN {X 0,Y 368.86,Z 292.162,A -85,B 0,C 180,E1 -12627.213,E2 -12627.213} C_VEL
LIN {X 0,Y 368.888,Z 292.155,A -85,B 0,C 180,E1 -12629.694,E2 -12629.694} C_VEL
LIN {X 0,Y 368.89,Z 292.157,A -85,B 0,C 180,E1 -12633.54,E2 -12633.54} C_VEL
LIN {X 0,Y 368.89,Z 292.155,A -85,B 0,C 180,E1 -12636.856,E2 -12636.856} C_VEL
LIN {X 0,Y 368.88,Z 292.162,A -85,B 0,C 180,E1 -12640.376,E2 -12640.376} C_VEL
LIN {X 0,Y 368.875,Z 292.159,A -85,B 0,C 180,E1 -12643.617,E2 -12643.617} C_VEL
LIN {X 0,Y 368.881,Z 292.161,A -85,B 0,C 180,E1 -12646.697,E2 -12646.697} C_VEL
LIN {X 0,Y 368.883,Z 292.161,A -85,B 0,C 180,E1 -12649.65,E2 -12649.65} C_VEL
LIN {X 0,Y 368.901,Z 292.203,A -85,B 0,C 180,E1 -12652.789,E2 -12652.789} C_VEL
LIN {X 0,Y 371.907,Z 302.593,A -85,B 0,C 180,E1 -12655.466,E2 -12655.466} C_VEL
LIN {X 0,Y 375.385,Z 316.012,A -85,B 0,C 180,E1 -12658.626,E2 -12658.626} C_VEL
LIN {X 0,Y 382.124,Z 331.146,A -85,B 0,C 180,E1 -12659.642,E2 -12659.642} C_VEL
LIN {X 0,Y 386.572,Z 354.671,A -85,B 0,C 180,E1 -12660.587,E2 -12660.587} C_VEL
LIN {X 0,Y 387.201,Z 358.774,A -85,B 0,C 180,E1 -12660.735,E2 -12660.735} C_VEL
LIN {X 0,Y 383.714,Z 482.568,A -85,B 0,C 180,E1 -12663.192,E2 -12663.192} C_VEL
LIN {X 0,Y 382.72,Z 498.402,A -85,B 0,C 180,E1 -12663.705,E2 -12663.705} C_VEL
LIN {X 0,Y 381.439,Z 513.314,A -85,B 0,C 180,E1 -12664.402,E2 -12664.402} C_VEL
LIN {X 0,Y 379.898,Z 527.842,A -85,B 0,C 180,E1 -12665.305,E2 -12665.305} C_VEL
LIN {X 0,Y 378.185,Z 542.242,A -85,B 0,C 180,E1 -12666.451,E2 -12666.451} C_VEL
LIN {X 0,Y 376.294,Z 555.708,A -85,B 0,C 180,E1 -12667.778,E2 -12667.778} C_VEL
LIN {X 0,Y 374.514,Z 567.993,A -85,B 0,C 180,E1 -12669.257,E2 -12669.257} C_VEL
LIN {X 0,Y 372.982,Z 578.636,A -85,B 0,C 180,E1 -12670.795,E2 -12670.795} C_VEL
LIN {X 0,Y 371.317,Z 589.429,A -85,B 0,C 180,E1 -12672.657,E2 -12672.657} C_VEL
LIN {X 0,Y 370.032,Z 598.628,A -85,B 0,C 180,E1 -12674.58,E2 -12674.58} C_VEL
LIN {X 0,Y 368.929,Z 607.305,A -85,B 0,C 180,E1 -12676.786,E2 -12676.786} C_VEL
LIN {X 0,Y 368.143,Z 614.279,A -85,B 0,C 180,E1 -12678.995,E2 -12678.995} C_VEL
LIN {X 0,Y 367.701,Z 619.763,A -85,B 0,C 180,E1 -12681.205,E2 -12681.205} C_VEL
LIN {X 0,Y 367.467,Z 623.9,A -85,B 0,C 180,E1 -12683.411,E2 -12683.411} C_VEL
LIN {X 0,Y 367.384,Z 626.785,A -85,B 0,C 180,E1 -12685.612,E2 -12685.612} C_VEL
LIN {X 0,Y 367.353,Z 628.48,A -85,B 0,C 180,E1 -12687.808,E2 -12687.808} C_VEL
LIN {X 0,Y 367.457,Z 629.024,A -85,B 0,C 180,E1 -12690,E2 -12690} C_VEL
LIN {X 0,Y 367.354,Z 628.382,A -85,B 0,C 180,E1 -12692.193,E2 -12692.193} C_VEL
LIN {X 0,Y 367.39,Z 626.532,A -85,B 0,C 180,E1 -12694.389,E2 -12694.389} C_VEL
LIN {X 0,Y 367.484,Z 623.481,A -85,B 0,C 180,E1 -12696.589,E2 -12696.589} C_VEL
LIN {X 0,Y 367.702,Z 619.156,A -85,B 0,C 180,E1 -12698.796,E2 -12698.796} C_VEL
LIN {X 0,Y 368.135,Z 613.443,A -85,B 0,C 180,E1 -12701.006,E2 -12701.006} C_VEL
LIN {X 0,Y 368.906,Z 606.191,A -85,B 0,C 180,E1 -12703.215,E2 -12703.215} C_VEL
LIN {X 0,Y 369.814,Z 598.423,A -85,B 0,C 180,E1 -12705.148,E2 -12705.148} C_VEL
LIN {X 0,Y 370.948,Z 589.068,A -85,B 0,C 180,E1 -12707.077,E2 -12707.077} C_VEL
LIN {X 0,Y 372.427,Z 579.568,A -85,B 0,C 180,E1 -12708.712,E2 -12708.712} C_VEL
LIN {X 0,Y 373.876,Z 568.257,A -85,B 0,C 180,E1 -12710.35,E2 -12710.35} C_VEL
LIN {X 0,Y 375.513,Z 555.853,A -85,B 0,C 180,E1 -12711.837,E2 -12711.837} C_VEL
LIN {X 0,Y 377.281,Z 542.18,A -85,B 0,C 180,E1 -12713.173,E2 -12713.173} C_VEL
LIN {X 0,Y 378.854,Z 528.061,A -85,B 0,C 180,E1 -12714.286,E2 -12714.286} C_VEL
LIN {X 0,Y 380.221,Z 513.983,A -85,B 0,C 180,E1 -12715.159,E2 -12715.159} C_VEL
LIN {X 0,Y 381.432,Z 498.549,A -85,B 0,C 180,E1 -12715.877,E2 -12715.877} C_VEL
LIN {X 0,Y 382.311,Z 483.406,A -85,B 0,C 180,E1 -12716.363,E2 -12716.363} C_VEL
LIN {X 0,Y 385.505,Z 358.655,A -85,B 0,C 180,E1 -12718.804,E2 -12718.804} C_VEL
LIN {X 0,Y 380.558,Z 331.548,A -85,B 0,C 180,E1 -12719.774,E2 -12719.774} C_VEL
LIN {X 0,Y 379.481,Z 327.161,A -85,B 0,C 180,E1 -12719.957,E2 -12719.957} C_VEL
LIN {X 0,Y 375.127,Z 316.713,A -85,B 0,C 180,E1 -12720.571,E2 -12720.571} C_VEL
LIN {X 0,Y 371.673,Z 302.614,A -85,B 0,C 180,E1 -12723.694,E2 -12723.694} C_VEL
LIN {X 0,Y 368.932,Z 292.156,A -85,B 0,C 180,E1 -12726.144,E2 -12726.144} C_VEL
LIN {X 0,Y 368.875,Z 292.165,A -85,B 0,C 180,E1 -12728.956,E2 -12728.956} C_VEL
LIN {X 0,Y 368.86,Z 292.166,A -85,B 0,C 180,E1 -12732.004,E2 -12732.004} C_VEL
LIN {X 0,Y 368.874,Z 292.162,A -85,B 0,C 180,E1 -12735.173,E2 -12735.173} C_VEL
LIN {X 0,Y 368.862,Z 292.169,A -85,B 0,C 180,E1 -12738.173,E2 -12738.173} C_VEL
LIN {X 0,Y 368.876,Z 292.156,A -85,B 0,C 180,E1 -12741.365,E2 -12741.365} C_VEL
LIN {X 0,Y 368.93,Z 292.145,A -85,B 0,C 180,E1 -12745.144,E2 -12745.144} C_VEL
LIN {X 0,Y 368.913,Z 292.154,A -85,B 0,C 180,E1 -12749.044,E2 -12749.044} C_VEL
LIN {X 0,Y 368.906,Z 292.159,A -85,B 0,C 180,E1 -12751.556,E2 -12751.556} C_VEL
LIN {X 0,Y 368.896,Z 292.161,A -85,B 0,C 180,E1 -12755.219,E2 -12755.219} C_VEL
LIN {X 0,Y 368.895,Z 292.161,A -85,B 0,C 180,E1 -12757.601,E2 -12757.601} C_VEL
LIN {X 0,Y 368.952,Z 292.149,A -85,B 0,C 180,E1 -12761.104,E2 -12761.104} C_VEL
LIN {X 0,Y 368.993,Z 292.141,A -85,B 0,C 180,E1 -12764.533,E2 -12764.533} C_VEL
LIN {X 0,Y 369.054,Z 292.113,A -85,B 0,C 180,E1 -12766.788,E2 -12766.788} C_VEL
LIN {X 0,Y 369.052,Z 292.136,A -85,B 0,C 180,E1 -12770.13,E2 -12770.13} C_VEL
LIN {X 0,Y 369.149,Z 292.126,A -85,B 0,C 180,E1 -12773.439,E2 -12773.439} C_VEL
LIN {X 0,Y 369.285,Z 292.088,A -85,B 0,C 180,E1 -12777.817,E2 -12777.817} C_VEL
LIN {X 0,Y 369.297,Z 292.106,A -85,B 0,C 180,E1 -12782.179,E2 -12782.179} C_VEL
LIN {X 0,Y 369.122,Z 292.098,A -85,B 0,C 180,E1 -12786.558,E2 -12786.558} C_VEL
LIN {X 0,Y 369.022,Z 292.141,A -85,B 0,C 180,E1 -12789.867,E2 -12789.867} C_VEL
LIN {X 0,Y 369.029,Z 292.134,A -85,B 0,C 180,E1 -12793.77,E2 -12793.77} C_VEL
LIN {X 0,Y 368.969,Z 292.124,A -85,B 0,C 180,E1 -12797.755,E2 -12797.755} C_VEL
LIN {X 0,Y 368.9,Z 292.157,A -85,B 0,C 180,E1 -12801.219,E2 -12801.219} C_VEL
LIN {X 0,Y 368.897,Z 292.151,A -85,B 0,C 180,E1 -12803.872,E2 -12803.872} C_VEL
LIN {X 0,Y 368.845,Z 292.137,A -85,B 0,C 180,E1 -12807.21,E2 -12807.21} C_VEL
LIN {X 0,Y 368.881,Z 292.154,A -85,B 0,C 180,E1 -12809.691,E2 -12809.691} C_VEL
LIN {X 0,Y 368.883,Z 292.161,A -85,B 0,C 180,E1 -12813.041,E2 -12813.041} C_VEL
LIN {X 0,Y 368.898,Z 292.135,A -85,B 0,C 180,E1 -12816.196,E2 -12816.196} C_VEL
LIN {X 0,Y 368.86,Z 292.153,A -85,B 0,C 180,E1 -12818.955,E2 -12818.955} C_VEL
LIN {X 0,Y 368.856,Z 292.161,A -85,B 0,C 180,E1 -12822.006,E2 -12822.006} C_VEL
LIN {X 0,Y 368.861,Z 292.144,A -85,B 0,C 180,E1 -12825.174,E2 -12825.174} C_VEL
LIN {X 0,Y 368.866,Z 292.16,A -85,B 0,C 180,E1 -12828.176,E2 -12828.176} C_VEL
LIN {X 0,Y 368.891,Z 292.152,A -85,B 0,C 180,E1 -12831.359,E2 -12831.359} C_VEL
LIN {X 0,Y 368.92,Z 292.155,A -85,B 0,C 180,E1 -12835.145,E2 -12835.145} C_VEL
LIN {X 0,Y 368.897,Z 292.146,A -85,B 0,C 180,E1 -12839.044,E2 -12839.044} C_VEL
LIN {X 0,Y 368.946,Z 292.155,A -85,B 0,C 180,E1 -12842.795,E2 -12842.795} C_VEL
LIN {X 0,Y 368.916,Z 292.151,A -85,B 0,C 180,E1 -12846.116,E2 -12846.116} C_VEL
LIN {X 0,Y 368.913,Z 292.149,A -85,B 0,C 180,E1 -12849.946,E2 -12849.946} C_VEL
LIN {X 0,Y 368.958,Z 292.144,A -85,B 0,C 180,E1 -12853.398,E2 -12853.398} C_VEL
LIN {X 0,Y 369.043,Z 292.137,A -85,B 0,C 180,E1 -12856.79,E2 -12856.79} C_VEL
LIN {X 0,Y 369.055,Z 292.135,A -85,B 0,C 180,E1 -12860.131,E2 -12860.131} C_VEL
LIN {X 0,Y 369.144,Z 292.125,A -85,B 0,C 180,E1 -12862.341,E2 -12862.341} C_VEL
LIN {X 0,Y 369.123,Z 292.13,A -85,B 0,C 180,E1 -12864.537,E2 -12864.537} C_VEL
LIN {X 0,Y 369.256,Z 292.215,A -85,B 0,C 180,E1 -12867.648,E2 -12867.648} C_VEL
LIN {X 0,Y 370.751,Z 298.206,A -85,B 0,C 180,E1 -12869.151,E2 -12869.151} C_VEL
LIN {X 0,Y 380.428,Z 319.849,A -85,B 0,C 180,E1 -12870.444,E2 -12870.444} C_VEL
LIN {X 0,Y 385.821,Z 332.651,A -85,B 0,C 180,E1 -12871.146,E2 -12871.146} C_VEL
LIN {X 0,Y 383.198,Z 440.904,A -85,B 0,C 180,E1 -12873.252,E2 -12873.252} C_VEL
LIN {X 0,Y 382.52,Z 464.687,A -85,B 0,C 180,E1 -12873.752,E2 -12873.752} C_VEL
LIN {X 0,Y 381.671,Z 480.047,A -85,B 0,C 180,E1 -12874.274,E2 -12874.274} C_VEL
LIN {X 0,Y 380.643,Z 494.55,A -85,B 0,C 180,E1 -12874.976,E2 -12874.976} C_VEL
LIN {X 0,Y 379.419,Z 508.303,A -85,B 0,C 180,E1 -12875.847,E2 -12875.847} C_VEL
LIN {X 0,Y 377.962,Z 522.032,A -85,B 0,C 180,E1 -12876.941,E2 -12876.941} C_VEL
LIN {X 0,Y 376.347,Z 535.202,A -85,B 0,C 180,E1 -12878.237,E2 -12878.237} C_VEL
LIN {X 0,Y 374.734,Z 547.533,A -85,B 0,C 180,E1 -12879.717,E2 -12879.717} C_VEL
LIN {X 0,Y 373.351,Z 557.638,A -85,B 0,C 180,E1 -12881.172,E2 -12881.172} C_VEL
LIN {X 0,Y 372.101,Z 561.765,A -85,B 0,C 180,E1 -12881.794,E2 -12881.794} C_VEL
LIN {X 0,Y 368.348,Z 568.223,A -85,B 0,C 180,E1 -12882.808,E2 -12882.808} C_VEL
LIN {X 0,Y 364.689,Z 574.33,A -85,B 0,C 180,E1 -12883.898,E2 -12883.898} C_VEL
LIN {X 0,Y 363.601,Z 577.714,A -85,B 0,C 180,E1 -12884.631,E2 -12884.631} C_VEL
LIN {X 0,Y 362.526,Z 585.518,A -85,B 0,C 180,E1 -12886.615,E2 -12886.615} C_VEL
LIN {X 0,Y 361.688,Z 592.239,A -85,B 0,C 180,E1 -12888.699,E2 -12888.699} C_VEL
LIN {X 0,Y 361.031,Z 597.858,A -85,B 0,C 180,E1 -12890.878,E2 -12890.878} C_VEL
LIN {X 0,Y 360.66,Z 601.99,A -85,B 0,C 180,E1 -12892.937,E2 -12892.937} C_VEL
LIN {X 0,Y 360.263,Z 605.514,A -85,B 0,C 180,E1 -12895.414,E2 -12895.414} C_VEL
LIN {X 0,Y 360.084,Z 607.602,A -85,B 0,C 180,E1 -12897.931,E2 -12897.931} C_VEL
LIN {X 0,Y 360.036,Z 608.103,A -85,B 0,C 180,E1 -12899.208,E2 -12899.208} C_VEL
LIN {X 0,Y 360.036,Z 608.19,A -85,B 0,C 180,E1 -12900.813,E2 -12900.813} C_VEL
LIN {X 0,Y 360.157,Z 607.32,A -85,B 0,C 180,E1 -12903.118,E2 -12903.118} C_VEL
LIN {X 0,Y 360.342,Z 605.709,A -85,B 0,C 180,E1 -12905.005,E2 -12905.005} C_VEL
LIN {X 0,Y 360.821,Z 601.67,A -85,B 0,C 180,E1 -12907.845,E2 -12907.845} C_VEL
LIN {X 0,Y 361.344,Z 597.434,A -85,B 0,C 180,E1 -12909.927,E2 -12909.927} C_VEL
LIN {X 0,Y 362.006,Z 592.233,A -85,B 0,C 180,E1 -12911.925,E2 -12911.925} C_VEL
LIN {X 0,Y 363.045,Z 584.94,A -85,B 0,C 180,E1 -12914.177,E2 -12914.177} C_VEL
LIN {X 0,Y 364.323,Z 576.917,A -85,B 0,C 180,E1 -12916.184,E2 -12916.184} C_VEL
LIN {X 0,Y 365.777,Z 568.001,A -85,B 0,C 180,E1 -12918.035,E2 -12918.035} C_VEL
LIN {X 0,Y 367.551,Z 557.22,A -85,B 0,C 180,E1 -12919.891,E2 -12919.891} C_VEL
LIN {X 0,Y 369.313,Z 545.998,A -85,B 0,C 180,E1 -12921.497,E2 -12921.497} C_VEL
LIN {X 0,Y 371.119,Z 534.1,A -85,B 0,C 180,E1 -12922.912,E2 -12922.912} C_VEL
LIN {X 0,Y 372.816,Z 521.524,A -85,B 0,C 180,E1 -12924.152,E2 -12924.152} C_VEL
LIN {X 0,Y 374.484,Z 507.459,A -85,B 0,C 180,E1 -12925.271,E2 -12925.271} C_VEL
LIN {X 0,Y 375.895,Z 493.247,A -85,B 0,C 180,E1 -12926.16,E2 -12926.16} C_VEL
LIN {X 0,Y 377.027,Z 478.711,A -85,B 0,C 180,E1 -12926.848,E2 -12926.848} C_VEL
LIN {X 0,Y 377.898,Z 463.441,A -85,B 0,C 180,E1 -12927.349,E2 -12927.349} C_VEL
LIN {X 0,Y 381.601,Z 336.218,A -85,B 0,C 180,E1 -12929.927,E2 -12929.927} C_VEL
LIN {X 0,Y 374.176,Z 319.864,A -85,B 0,C 180,E1 -12931.04,E2 -12931.04} C_VEL
LIN {X 0,Y 366.066,Z 303.892,A -85,B 0,C 180,E1 -12932.294,E2 -12932.294} C_VEL
LIN {X 0,Y 363.709,Z 299.651,A -85,B 0,C 180,E1 -12932.677,E2 -12932.677} C_VEL
LIN {X 0,Y 361.91,Z 293.029,A -85,B 0,C 180,E1 -12934.634,E2 -12934.634} C_VEL
LIN {X 0,Y 361.877,Z 293.032,A -85,B 0,C 180,E1 -12938.349,E2 -12938.349} C_VEL
LIN {X 0,Y 361.954,Z 293.027,A -85,B 0,C 180,E1 -12942.063,E2 -12942.063} C_VEL
LIN {X 0,Y 361.985,Z 293.02,A -85,B 0,C 180,E1 -12946.103,E2 -12946.103} C_VEL
LIN {X 0,Y 362.018,Z 293.015,A -85,B 0,C 180,E1 -12949.94,E2 -12949.94} C_VEL
LIN {X 0,Y 362.15,Z 292.997,A -85,B 0,C 180,E1 -12953.315,E2 -12953.315} C_VEL
LIN {X 0,Y 362.269,Z 292.984,A -85,B 0,C 180,E1 -12957.778,E2 -12957.778} C_VEL
LIN {X 0,Y 362.416,Z 292.964,A -85,B 0,C 180,E1 -12960.002,E2 -12960.002} C_VEL
LIN {X 0,Y 362.268,Z 292.979,A -85,B 0,C 180,E1 -12962.225,E2 -12962.225} C_VEL
LIN {X 0,Y 362.132,Z 293.003,A -85,B 0,C 180,E1 -12966.689,E2 -12966.689} C_VEL
LIN {X 0,Y 361.991,Z 293.018,A -85,B 0,C 180,E1 -12970.065,E2 -12970.065} C_VEL
LIN {X 0,Y 361.99,Z 293.014,A -85,B 0,C 180,E1 -12973.9,E2 -12973.9} C_VEL
LIN {X 0,Y 361.92,Z 293.023,A -85,B 0,C 180,E1 -12976.936,E2 -12976.936} C_VEL
LIN {X 0,Y 361.876,Z 293.03,A -85,B 0,C 180,E1 -12980.463,E2 -12980.463} C_VEL
LIN {X 0,Y 361.855,Z 293.033,A -85,B 0,C 180,E1 -12984.103,E2 -12984.103} C_VEL
LIN {X 0,Y 361.835,Z 293.037,A -85,B 0,C 180,E1 -12987.787,E2 -12987.787} C_VEL
LIN {X 0,Y 361.821,Z 293.034,A -85,B 0,C 180,E1 -12991.281,E2 -12991.281} C_VEL
LIN {X 0,Y 361.846,Z 293.032,A -85,B 0,C 180,E1 -12994.283,E2 -12994.283} C_VEL
LIN {X 0,Y 361.852,Z 293.032,A -85,B 0,C 180,E1 -12997.223,E2 -12997.223} C_VEL
LIN {X 0,Y 361.806,Z 293.04,A -85,B 0,C 180,E1 -13000.752,E2 -13000.752} C_VEL
LIN {X 0,Y 361.808,Z 293.043,A -85,B 0,C 180,E1 -13004.371,E2 -13004.371} C_VEL
LIN {X 0,Y 361.82,Z 293.039,A -85,B 0,C 180,E1 -13007.572,E2 -13007.572} C_VEL
LIN {X 0,Y 361.841,Z 293.042,A -85,B 0,C 180,E1 -13011.573,E2 -13011.573} C_VEL
LIN {X 0,Y 361.877,Z 293.236,A -85,B 0,C 180,E1 -13012.128,E2 -13012.128} C_VEL
LIN {X 0,Y 365.058,Z 304.057,A -85,B 0,C 180,E1 -13015.022,E2 -13015.022} C_VEL
